# B&R Automation Studio project Panasonic_LinkaKapacitorov_A2021040 (part 5)

#### Main.st - Init, cyclic, exit code
```iecst
PROGRAM _INIT
	(* Insert code here *)

END_PROGRAM

PROGRAM _CYCLIC

	//Volanie podprogramov//
	OvlCentrovacky;

	//Volanie funkcie SequenceControl//
	SequenceControl(SC:= SC_StoperDopravNG);

	//Príznak obsluha potvrdila paletku NG na dopravníku NG//
	IF StoperDopravNG.Automat AND StoperDopravNG.STAV.PaletkaNaKonciDopravnika_NG AND Vizu.TL_NavratPaletkyNG THEN
		StoperDopravNG.STAV.ObsluhaPotvrdilaPaletkuNG:= TRUE;
		Vizu.TL_NavratPaletkyNG:= FALSE;
	END_IF
	IF NOT StoperDopravNG.IN.Dopravnik_PritomnostPaletky_OS4 THEN
		StoperDopravNG.STAV.ObsluhaPotvrdilaPaletkuNG:= FALSE;
	END_IF

	//Zmena farby tlačítka potvrdenie návratu paletky NG//
	IF StoperDopravNG.STAV.ObsluhaPotvrdilaPaletkuNG THEN
		Vizu.FarbaTlacitka_PotvrdPaletkuNG:= Blikac500ms;
	ELSE
		Vizu.FarbaTlacitka_PotvrdPaletkuNG:= TRUE;
	END_IF

	//Zobrazenie hlásenia potvrd paletku NG//
	IF StoperDopravNG.STAV.PaletkaNaKonciDopravnika_NG AND NOT StoperDopravNG.STAV.DopravnikNG_BUSY AND StoperDopravNG.STAV.PoINIT THEN
		Vizu.ZobrazHlasenie_PotvrdPaletkyNG:= 0;
	ELSE
		Vizu.ZobrazHlasenie_PotvrdPaletkyNG:= 1;
	END_IF

	//Príznak paletka NG na konci dopravníka//
	IF StoperDopravNG.Automat AND StoperDopravNG.IN.Dopravnik_PritomnostPaletky_OS4 THEN
		StoperDopravNG.STAV.PaletkaNaKonciDopravnika_NG:= TRUE;
	END_IF

	//Zamknutie tlačítka potvrdenie paletky NG//
	IF StoperDopravNG.STAV.PaletkaNaKonciDopravnika_NG AND StoperDopravNG.IN.Dopravnik_PritomnostPaletky_OS4 THEN
		Vizu.TL_PotvrdeniePaletky_NG_DISABLE:= FALSE;
	ELSE
		Vizu.TL_PotvrdeniePaletky_NG_DISABLE:= TRUE;
	END_IF

	//Zamknutie tlačítka zrušenie paletky NG//
	IF StoperDopravNG.STAV.PaletkaNaKonciDopravnika_NG AND NOT StoperDopravNG.IN.Dopravnik_PritomnostPaletky_OS4 THEN
		Vizu.TL_ZruseniePaletky_NG_DISABLE:= FALSE;
	ELSE
		Vizu.TL_ZruseniePaletky_NG_DISABLE:= TRUE;
	END_IF

	//Zrušenie paletky NG//
	IF StoperDopravNG.STAV.ObsluhaPotvrdilaZrusPaletkyNG THEN
		StoperDopravNG.STAV.PaletkaNaKonciDopravnika_NG:= FALSE;
		StoperDopravNG.STAV.ObsluhaPotvrdilaZrusPaletkyNG:= FALSE;
	END_IF

	//Reset sekcie //
	IF StoperDopravNG.Reset THEN
		SC_StoperDopravNG.Step:= 0;
		StoperDopravNG.Reset:= FALSE;
	ELSIF NOT Safety.STAV.ZonaCS_AKTIVNA THEN
		SC_StoperDopravNG.Step:= 0;
	END_IF

	CASE SC_StoperDopravNG.Step OF

		0:
			SC_StoperDopravNG.StepName:='0 - Nulovanie';
			StoperDopravNG.Automat:= FALSE;
			StoperDopravNG.KoniecCyklu:= FALSE;
			StoperDopravNG.Manual:= FALSE;
			StoperDopravNG.STAV.PoINIT:= FALSE;
			StoperDopravNG.OUT.Dopravnik_ChodVPRED_ELR3:= FALSE;
			StoperDopravNG.OUT.Dopravnik_ChodVZAD_ELR3:= FALSE;
			SC_OvlCentrovacky.Step:= 0;
			StoperDopravNG.STAV.ObsluhaPotvrdilaPaletkuNG:= FALSE;
			StoperDopravNG.RR_Dopravnik_VPRED:= FALSE;
			StoperDopravNG.RR_Dopravnik_VZAD:= FALSE;
			Vizu.ZobrazHlasenie_PotvrdPaletkyNG:= 1;
			StoperDopravNG.STAV.PrebiehaVyvazaniePaletky:= FALSE;
			StoperDopravNG.STAV.PaletkaNaKonciDopravnika_NG:= FALSE;
			StoperDopravNG.STAV.DopravnikNG_BUSY:= FALSE;
			StoperDopravNG_Statistika.IN.START_MeraniaCasu:= FALSE;

			IF Safety.STAV.ZonaCS_AKTIVNA AND Safety.STAV.ZonaBunky_AKTIVNA AND Linka.IN.TlakVzduchu_OK_S2 AND NOT NastalaPorucha AND Linka.STAV.Hardware_OK THEN
				SC_StoperDopravNG.ResetStep:= TRUE;
				SC_StoperDopravNG.Step:= 1;
			END_IF

		1:
			SC_StoperDopravNG.StepName:='1 - Cakam na spustenie vyroby';
			StoperDopravNG.KoniecCyklu:= FALSE;
			IF StoperDopravNG.Automat THEN
				SC_StoperDopravNG.Step:= 2;
			ELSIF StoperDopravNG.Manual THEN
				SC_StoperDopravNG.Step:= 700;
			END_IF

			//********************************************************Inicializácia****************************************************************************//

		2:
			SC_StoperDopravNG.StepName:='2 - Inicializacia - cakam na spustenie inicializacie';
			SC_StoperDopravNG.IdleTime.PT:= T#4s;
			SC_StoperDopravNG.AlarmTime.PT:= T#5s;

			IF DopravBunky.STAV.PoINIT AND Robot.STAV.PoINIT THEN
				SC_StoperDopravNG.ResetStep:= TRUE;
				SC_StoperDopravNG.Step:= 5;
			END_IF

		5:
			SC_StoperDopravNG.StepName:='5 - Inicializacia - hladanie paletky na dopravniku NG';
			SC_StoperDopravNG.IdleTime.PT:= T#5s;
			SC_StoperDopravNG.AlarmTime.PT:= T#5s;

			IF NOT SC_StoperDopravNG.Switch1 AND Safety.STAV.MutingRobota_AKTIVNY THEN
				StoperDopravNG.OUT.Dopravnik_ChodVPRED_ELR3:= TRUE;
				StoperDopravNG.STAV.DopravnikNG_BUSY:= TRUE;
				SC_StoperDopravNG.IdleTime.IN:= TRUE;
				SC_StoperDopravNG.Switch1:= TRUE;
			END_IF

			IF StoperDopravNG.IN.Dopravnik_PritomnostPaletky_OS4 THEN
				StoperDopravNG.OUT.Dopravnik_ChodVPRED_ELR3:= FALSE;
				StoperDopravNG.STAV.DopravnikNG_BUSY:= FALSE;
				Vizu.ZobrazHlasenie_PotvrdPaletkyNG:= 0;
				SC_StoperDopravNG.ResetStep:= TRUE;
				SC_StoperDopravNG.Step:= 10;
			ELSIF SC_StoperDopravNG.IdleTime.Q THEN
				StoperDopravNG.OUT.Dopravnik_ChodVPRED_ELR3:= FALSE;
				StoperDopravNG.STAV.DopravnikNG_BUSY:= FALSE;
				SC_StoperDopravNG.ResetStep:= TRUE;
				SC_StoperDopravNG.Step:= 10;
			END_IF

		10:
			SC_StoperDopravNG.StepName:='10 - Inicializacia - presun centrovacky do sterdnej polohy';
			SC_StoperDopravNG.IdleTime.PT:= T#4s;
			SC_StoperDopravNG.AlarmTime.PT:= T#5s;

			IF NOT SC_StoperDopravNG.Switch1 THEN
				Centrovacku_VYSTRED:= TRUE;
				SC_StoperDopravNG.Switch1:= TRUE;
			END_IF

			IF StoperDopravNG.IN.Centrovanie_StrednaPoloha_IS20 THEN
				SC_StoperDopravNG.ResetStep:= TRUE;
				SC_StoperDopravNG.Step:= 13;
			END_IF

		13:
			SC_StoperDopravNG.StepName:='13 - Inicializacia - hladanie paletky';
			SC_StoperDopravNG.IdleTime.PT:= T#3s;
			SC_StoperDopravNG.AlarmTime.PT:= T#7s;

			SC_StoperDopravNG.IdleTime.IN:= StoperDopravNG.IN.Stoper_PritomnostPaletky_IS15;
			SC_StoperDopravNG.AlarmTime.IN:= TRUE;

			IF SC_StoperDopravNG.IdleTime.Q THEN
				StoperDopravNG.STAV.PoINIT:= TRUE;
				SC_StoperDopravNG.ResetStep:= TRUE;
				SC_StoperDopravNG.Step:= 100;
			ELSIF SC_StoperDopravNG.AlarmTime.Q AND NOT StoperDopravNG.IN.Stoper_PritomnostPaletky_IS15 THEN
				StoperDopravNG.STAV.PoINIT:= TRUE;
				SC_StoperDopravNG.ResetStep:= TRUE;
				SC_StoperDopravNG.Step:= 100;
			END_IF

			//********************************************************Automatický režim****************************************************************************//

		100:
			SC_StoperDopravNG.StepName:='100 - Automaticky Rezim - cakam na príchod paletky na stoper';
			SC_StoperDopravNG.IdleTime.PT:= T#3s;
			SC_StoperDopravNG.AlarmTime.PT:= T#5s;

			SC_StoperDopravNG.IdleTime.IN:= StoperDopravNG.IN.Stoper_PritomnostPaletky_IS15;

			IF StoperDopravNG.KoniecCyklu THEN
				SC_StoperDopravNG.ResetStep:= TRUE;
				SC_StoperDopravNG.Step:= 0;
			ELSIF SC_StoperDopravNG.IdleTime.Q THEN
				StoperDopravNG_Statistika.IN.START_MeraniaCasu:= TRUE;
				StoperDopravNG_Statistika.IN.ZAPIS_MeraniaCasu:= TRUE;
				SC_StoperDopravNG.ResetStep:= TRUE;
				SC_StoperDopravNG.Step:= 110;
			ELSIF NOT StoperDopravNG.IN.Stoper_PritomnostPaletky_IS15 AND StoperDopravNG.IN.Dopravnik_PritomnostPaletky_OS4 AND NOT StoperEtiketovania.STAV.PrebiehaVyvazaniePaletky AND StoperDopravNG.STAV.ObsluhaPotvrdilaPaletkuNG AND NOT StoperEtiketovania.STAV.Etiketovanie_BUSY AND NOT StoperVystupDopravnika.IN.ZaplnenieBuffera_IS28 THEN
				StoperDopravNG.STAV.DopravnikNG_BUSY:= TRUE;
				SC_StoperDopravNG.ResetStep:= TRUE;
				SC_StoperDopravNG.Step:= 150;
			END_IF

		110:
			SC_StoperDopravNG.StepName:='110 - Automaticky Rezim - kontrola stavu paletky';
			SC_StoperDopravNG.IdleTime.PT:= T#200ms;
			SC_StoperDopravNG.AlarmTime.PT:= T#10s;

			IF StoperEtiketovania.STAV.VyvazamPaletkuNG THEN
				StoperDopravNG.STAV.DopravnikNG_BUSY:= TRUE;
				SC_StoperDopravNG.ResetStep:= TRUE;
				SC_StoperDopravNG.Step:= 120;
			ELSE
				SC_StoperDopravNG.ResetStep:= TRUE;
				SC_StoperDopravNG.Step:= 170;
			END_IF

			//Vyvezenie na dopravník NG//
		120:
			SC_StoperDopravNG.StepName:='120 - Automaticky Rezim - kontrola muting pozicie robota';
			SC_StoperDopravNG.IdleTime.PT:= T#200ms;
			SC_StoperDopravNG.AlarmTime.PT:= T#10s;

			IF Safety.STAV.MutingRobota_AKTIVNY AND Robot.STAV.PoINIT THEN
				SC_StoperDopravNG.ResetStep:= TRUE;
				SC_StoperDopravNG.Step:= 128;
			ELSIF NOT Safety.STAV.MutingRobota_AKTIVNY AND Robot.STAV.PoINIT THEN
				Robot.KOM_OUT.PresunDoMutingPozicie:= TRUE;
				SC_StoperDopravNG.ResetStep:= TRUE;
				SC_StoperDopravNG.Step:= 123;
			END_IF

		123:
			SC_StoperDopravNG.StepName:='123 - Automaticky Rezim - cakam na ukoncenie cinnosti robota';
			SC_StoperDopravNG.IdleTime.PT:= T#200ms;
			SC_StoperDopravNG.AlarmTime.PT:= T#10s;

			IF Robot.KOM_IN.Stav_RobotCinnostUkoncena THEN
				Robot.KOM_OUT.PresunDoMutingPozicie:= FALSE;
				SC_StoperDopravNG.ResetStep:= TRUE;
				SC_StoperDopravNG.Step:= 125;
			END_IF

		125:
			SC_StoperDopravNG.StepName:='125 - Automaticky Rezim - cakam na zrusenie signalu cinnost robota ukoncena';
			SC_StoperDopravNG.IdleTime.PT:= T#200ms;
			SC_StoperDopravNG.AlarmTime.PT:= T#5s;

			IF NOT Robot.KOM_IN.Stav_RobotCinnostUkoncena AND Safety.STAV.MutingRobota_AKTIVNY THEN
				SC_StoperDopravNG.ResetStep:= TRUE;
				SC_StoperDopravNG.Step:= 128;
			END_IF

		128:
			SC_StoperDopravNG.StepName:='128 - Automaticky Rezim - zdvih centrovacky pre vyvezenie paletky na dopravnik NG';
			SC_StoperDopravNG.IdleTime.PT:= T#200ms;
			SC_StoperDopravNG.AlarmTime.PT:= T#10s;

			IF NOT SC_StoperDopravNG.Switch1 THEN
				Centrovacku_VYSUN:= TRUE;
				SC_StoperDopravNG.Switch1:= TRUE;
			END_IF

			IF StoperDopravNG.IN.Centrovanie_HornaPoloha_IS19 THEN
				SC_StoperDopravNG.ResetStep:= TRUE;
				SC_StoperDopravNG.Step:= 130;
			END_IF

		130:
			SC_StoperDopravNG.StepName:='130 - Automaticky Rezim - spustenie dopravnika NG vpred';
			SC_StoperDopravNG.IdleTime.PT:= T#200ms;
			SC_StoperDopravNG.AlarmTime.PT:= T#10s;

			SC_StoperDopravNG.IdleTime.IN:= StoperDopravNG.IN.Dopravnik_PritomnostPaletky_OS4;

			IF NOT SC_StoperDopravNG.Switch1 AND Safety.STAV.MutingRobota_AKTIVNY THEN
				StoperDopravNG.OUT.Dopravnik_ChodVPRED_ELR3:= TRUE;
				SC_StoperDopravNG.AlarmTime.IN:= TRUE;
				SC_StoperDopravNG.Switch1:= TRUE;
			END_IF

			IF SC_StoperDopravNG.IdleTime.Q THEN
				(*StoperDopravNG.OUT.Dopravnik_ChodVPRED_ELR3:= FALSE;*)
				StoperDopravNG.STAV.PaletkaNaKonciDopravnika_NG:= TRUE;
				StoperDopravNG.STAV.DopravnikNG_BUSY:= FALSE;
				Vizu.ZobrazHlasenie_PotvrdPaletkyNG:= 0;
				SC_StoperDopravNG.ResetStep:= TRUE;
				SC_StoperDopravNG.Step:= 133;
			ELSIF SC_StoperDopravNG.AlarmTime.Q THEN
				Alarmy[63]:= TRUE;
				PoruchaBunky:= TRUE;
				SC_StoperDopravNG.ResetStep:= TRUE;
				SC_StoperDopravNG.Step:= 0;
			END_IF

		133:
			SC_StoperDopravNG.StepName:='133 - Automaticky Rezim - presun centrovacky do strednej polohy';
			SC_StoperDopravNG.IdleTime.PT:= T#4s;
			SC_StoperDopravNG.AlarmTime.PT:= T#5s;

			IF NOT SC_StoperDopravNG.Switch1 THEN
				Centrovacku_VYSTRED:= TRUE;
				SC_StoperDopravNG.Switch1:= TRUE;
			END_IF

			IF StoperDopravNG.IN.Centrovanie_StrednaPoloha_IS20 THEN
				SC_StoperDopravNG.ResetStep:= TRUE;
				SC_StoperDopravNG.Step:= 100;
			END_IF

			//Navezenie z dopravníka NG//
		150:
			SC_StoperDopravNG.StepName:='150 - Automaticky Rezim - kontrola muting pozicie robota';
			SC_StoperDopravNG.IdleTime.PT:= T#200ms;
			SC_StoperDopravNG.AlarmTime.PT:= T#10s;

			IF Safety.STAV.MutingRobota_AKTIVNY THEN
				SC_StoperDopravNG.ResetStep:= TRUE;
				SC_StoperDopravNG.Step:= 158;
			ELSIF NOT Safety.STAV.MutingRobota_AKTIVNY AND Robot.Automat THEN
				Robot.KOM_OUT.PresunDoMutingPozicie:= TRUE;
				SC_StoperDopravNG.ResetStep:= TRUE;
				SC_StoperDopravNG.Step:= 153;
			END_IF

		153:
			SC_StoperDopravNG.StepName:='153 - Automaticky Rezim - cakam na ukoncenie cinnosti robota';
			SC_StoperDopravNG.IdleTime.PT:= T#200ms;
			SC_StoperDopravNG.AlarmTime.PT:= T#10s;

			IF Robot.KOM_IN.Stav_RobotCinnostUkoncena THEN
				Robot.KOM_OUT.PresunDoMutingPozicie:= FALSE;
				SC_StoperDopravNG.ResetStep:= TRUE;
				SC_StoperDopravNG.Step:= 155;
			END_IF

		155:
			SC_StoperDopravNG.StepName:='155 - Automaticky Rezim - cakam na zrusenie signalu cinnost robota ukoncena';
			SC_StoperDopravNG.IdleTime.PT:= T#200ms;
			SC_StoperDopravNG.AlarmTime.PT:= T#5s;

			IF NOT Robot.KOM_IN.Stav_RobotCinnostUkoncena AND Safety.STAV.MutingRobota_AKTIVNY THEN
				SC_StoperDopravNG.ResetStep:= TRUE;
				SC_StoperDopravNG.Step:= 158;
			END_IF

		158:
			SC_StoperDopravNG.StepName:='150 - Automaticky Rezim - zdvih centrovacky pre navezenie paletky z dopravnika NG';
			SC_StoperDopravNG.IdleTime.PT:= T#200ms;
			SC_StoperDopravNG.AlarmTime.PT:= T#10s;

			IF NOT SC_StoperDopravNG.Switch1 THEN
				Centrovacku_VYSUN:= TRUE;
				SC_StoperDopravNG.Switch1:= TRUE;
			END_IF

			IF StoperDopravNG.IN.Centrovanie_HornaPoloha_IS19 THEN
				SC_StoperDopravNG.ResetStep:= TRUE;
				SC_StoperDopravNG.Step:= 160;
			END_IF

		160:
			SC_StoperDopravNG.StepName:='160 - Automaticky Rezim - spustenie dopravnika NG vzad';
			SC_StoperDopravNG.IdleTime.PT:= T#200ms;
			SC_StoperDopravNG.AlarmTime.PT:= T#10s;

			SC_StoperDopravNG.IdleTime.IN:= StoperDopravNG.IN.Stoper_PritomnostPaletky_IS15;

			IF NOT SC_StoperDopravNG.Switch1 AND Safety.STAV.MutingRobota_AKTIVNY THEN
				StoperDopravNG.OUT.Dopravnik_ChodVPRED_ELR3:= FALSE;
				StoperDopravNG.OUT.Dopravnik_ChodVZAD_ELR3:= TRUE;
				SC_StoperDopravNG.AlarmTime.IN:= TRUE;
				SC_StoperDopravNG.Switch1:= TRUE;
			END_IF

			IF SC_StoperDopravNG.IdleTime.Q THEN
				StoperDopravNG.STAV.PaletkaNaKonciDopravnika_NG:= FALSE;
				StoperDopravNG.OUT.Dopravnik_ChodVZAD_ELR3:= FALSE;
				StoperDopravNG.STAV.DopravnikNG_BUSY:= FALSE;
				SC_StoperDopravNG.ResetStep:= TRUE;
				SC_StoperDopravNG.Step:= 163;
			ELSIF SC_StoperDopravNG.AlarmTime.Q THEN
				Alarmy[64]:= TRUE;
				PoruchaBunky:= TRUE;
				SC_StoperDopravNG.ResetStep:= TRUE;
				SC_StoperDopravNG.Step:= 0;
			END_IF

		163:
			SC_StoperDopravNG.StepName:='163 - Automaticky Rezim - presun centrovacky do strednej polohy';
			SC_StoperDopravNG.IdleTime.PT:= T#4s;
			SC_StoperDopravNG.AlarmTime.PT:= T#5s;

			IF NOT SC_StoperDopravNG.Switch1 THEN
				Centrovacku_VYSTRED:= TRUE;
				SC_StoperDopravNG.Switch1:= TRUE;
			END_IF

			IF StoperDopravNG.IN.Centrovanie_StrednaPoloha_IS20 THEN
				SC_StoperDopravNG.ResetStep:= TRUE;
				SC_StoperDopravNG.Step:= 170;
			END_IF

			//Vyvezenie paletky na výstupný dopravník//
		170:
			SC_StoperDopravNG.StepName:='170 - Automaticky Rezim - cakam na vyvezenie na stoper vystupneho dopravnika';
			SC_StoperDopravNG.IdleTime.PT:= T#4s;
			SC_StoperDopravNG.AlarmTime.PT:= T#5s;

			IF StoperDopravNG.KoniecCyklu THEN
				SC_StoperDopravNG.ResetStep:= TRUE;
				SC_StoperDopravNG.Step:= 0;
			ELSIF NOT StoperVystupDopravnika.IN.ZaplnenieBuffera_IS28 AND VystupnyDopravnik.STAV.PoINIT THEN
				SC_StoperDopravNG.ResetStep:= TRUE;
				SC_StoperDopravNG.Step:= 173;
			END_IF

		173:
			SC_StoperDopravNG.StepName:='173 - Automaticky Rezim - vyvazam paletku na stoper vystupneho dopravnika';
			SC_StoperDopravNG.IdleTime.PT:= T#500ms;
			SC_StoperDopravNG.AlarmTime.PT:= T#10s;

			SC_StoperDopravNG.IdleTime.IN:= NOT StoperDopravNG.IN.Stoper_PritomnostPaletky_IS15;

			IF NOT SC_StoperDopravNG.Switch1 THEN
				Centrovacku_ZASUN:= TRUE;
				StoperDopravNG.STAV.PrebiehaVyvazaniePaletky:= TRUE;
				SC_StoperDopravNG.AlarmTime.IN:= TRUE;
				SC_StoperDopravNG.Switch1:= TRUE;
			END_IF

			IF NOT SC_StoperDopravNG.Switch2 AND SC_StoperDopravNG.IdleTime.Q AND SC_OvlCentrovacky.Step = 1 THEN
				Centrovacku_VYSTRED:= TRUE;
				SC_StoperDopravNG.AlarmTime.IN:= FALSE;
				SC_StoperDopravNG.Switch2:= TRUE;
			END_IF

			IF NOT Linka.Rezim_Priechodny AND StoperDopravNG.IN.Centrovanie_StrednaPoloha_IS20 AND NOT StoperDopravNG.IN.Stoper_PritomnostPaletky_IS15 THEN
				StoperDopravNG.STAV.PrebiehaVyvazaniePaletky:= FALSE;
				SC_StoperDopravNG.ResetStep:= TRUE;
				SC_StoperDopravNG.Step:= 100;
			ELSIF Linka.Rezim_Priechodny AND StoperDopravNG.IN.Centrovanie_StrednaPoloha_IS20 AND NOT StoperDopravNG.IN.Stoper_PritomnostPaletky_IS15 AND StoperVystupDopravnika.IN.ZaplnenieBuffera_IS28 THEN
				StoperDopravNG.STAV.PrebiehaVyvazaniePaletky:= FALSE;
				SC_StoperDopravNG.ResetStep:= TRUE;
				SC_StoperDopravNG.Step:= 100;
			ELSIF SC_StoperDopravNG.AlarmTime.Q THEN
				Alarmy[65]:= TRUE;
				PoruchaBunky:= TRUE;
				SC_StoperDopravNG.ResetStep:= TRUE;
				SC_StoperDopravNG.Step:= 0;
			END_IF

			//*******************************************************Manuálny režim*******************************************************************************//
		700:
			SC_StoperDopravNG.StepName:='700 - Manualny Rezim';
			SC_StoperDopravNG.IdleTime.PT:= T#8s;
			SC_StoperDopravNG.AlarmTime.PT:= T#5s;

			//Ovládanie dopravníka//
			IF StoperDopravNG.RR_Dopravnik_VPRED THEN
				StoperDopravNG.RR_Dopravnik_VZAD:= FALSE;
				StoperDopravNG.OUT.Dopravnik_ChodVZAD_ELR3:= FALSE;
				StoperDopravNG.OUT.Dopravnik_ChodVPRED_ELR3:= TRUE;
			ELSIF StoperDopravNG.RR_Dopravnik_VZAD THEN
				StoperDopravNG.RR_Dopravnik_VPRED:= FALSE;
				StoperDopravNG.OUT.Dopravnik_ChodVPRED_ELR3:= FALSE;
				StoperDopravNG.OUT.Dopravnik_ChodVZAD_ELR3:= TRUE;
			ELSE
				StoperDopravNG.OUT.Dopravnik_ChodVPRED_ELR3:= FALSE;
				StoperDopravNG.OUT.Dopravnik_ChodVZAD_ELR3:= FALSE;
			END_IF

	END_CASE

END_PROGRAM

PROGRAM _EXIT
	(* Insert code here *)

END_PROGRAM
```

#### Variables.var - Local variables
```iecst
VAR
	SC_OvlCentrovacky : SequenceControlTyp;
	Centrovacku_VYSUN : BOOL;
	Centrovacku_ZASUN : BOOL;
	Centrovacku_VYSTRED : BOOL := FALSE;
END_VAR
```

#### OvlCentrovacky.st
```iecst
ACTION OvlCentrovacky:

	//Volanie funkcie SequenceControl//
	SequenceControl(SC:= SC_OvlCentrovacky);

	CASE SC_OvlCentrovacky.Step OF

		0:
			SC_OvlCentrovacky.StepName:= '0 - Nulovanie';
			Centrovacku_VYSUN:= FALSE;
			Centrovacku_ZASUN:= FALSE;
			Centrovacku_VYSTRED:= FALSE;
			//			StoperDopravNG.OUT.Centrovanie_VYSUN_YV009:= FALSE;
			//			StoperDopravNG.OUT.Centrovanie_ZASUN_YV010:= FALSE;

			IF SC_StoperDopravNG.Step <> 0 THEN
				SC_OvlCentrovacky.ResetStep:= TRUE;
				SC_OvlCentrovacky.Step:= 1;
			END_IF

		1:
			SC_OvlCentrovacky.StepName:= '1 - Rozhodnutie o cinnosti';
			IF Centrovacku_VYSUN THEN
				SC_OvlCentrovacky.Step:= 10;
			ELSIF Centrovacku_ZASUN THEN
				SC_OvlCentrovacky.Step:= 20;
			ELSIF Centrovacku_VYSTRED THEN
				SC_OvlCentrovacky.Step:= 30;
			END_IF

		10:
			SC_OvlCentrovacky.StepName:= '10 - Vysunutie centrovacky hore';
			SC_OvlCentrovacky.IdleTime.PT:= T#3s;
			SC_OvlCentrovacky.AlarmTime.PT:= T#6s;

			IF StoperDopravNG.Automat THEN
				SC_OvlCentrovacky.AlarmTime.IN:= TRUE;
			ELSE
				SC_OvlCentrovacky.IdleTime.IN:= TRUE;
			END_IF

			IF NOT SC_OvlCentrovacky.Switch1 THEN
				StoperDopravNG.OUT.Centrovanie_ZASUN_YV010:= FALSE;
				StoperDopravNG.OUT.Centrovanie_VYSUN_YV009:= TRUE;
				SC_OvlCentrovacky.Switch1:= TRUE;
			END_IF

			IF StoperDopravNG.IN.Centrovanie_HornaPoloha_IS19 OR SC_OvlCentrovacky.IdleTime.Q THEN
				SC_OvlCentrovacky.ResetStep:= TRUE;
				SC_OvlCentrovacky.Step:= 0;
			ELSIF SC_OvlCentrovacky.AlarmTime.Q THEN
				Alarmy[57]:= TRUE;
				PoruchaBunky:= TRUE;
				SC_OvlCentrovacky.ResetStep:= TRUE;
				SC_OvlCentrovacky.Step:= 0;
			END_IF

		20:
			SC_OvlCentrovacky.StepName:= '20 - Zasunutie centrovacky dole';
			SC_OvlCentrovacky.IdleTime.PT:= T#3s;
			SC_OvlCentrovacky.AlarmTime.PT:= T#6s;

			IF StoperDopravNG.Automat THEN
				SC_OvlCentrovacky.AlarmTime.IN:= TRUE;
			ELSE
				SC_OvlCentrovacky.IdleTime.IN:= TRUE;
			END_IF

			IF NOT SC_OvlCentrovacky.Switch1 THEN
				StoperDopravNG.OUT.Centrovanie_VYSUN_YV009:= FALSE;
				StoperDopravNG.OUT.Centrovanie_ZASUN_YV010:= TRUE;
				SC_OvlCentrovacky.Switch1:= TRUE;
			END_IF

			IF StoperDopravNG.IN.Centrovanie_SpodnaPoloha_IS21 OR SC_OvlCentrovacky.IdleTime.Q THEN
				SC_OvlCentrovacky.ResetStep:= TRUE;
				SC_OvlCentrovacky.Step:= 0;
			ELSIF SC_OvlCentrovacky.AlarmTime.Q THEN
				Alarmy[58]:= TRUE;
				PoruchaBunky:= TRUE;
				SC_OvlCentrovacky.ResetStep:= TRUE;
				SC_OvlCentrovacky.Step:= 0;
			END_IF

		30:
			SC_OvlCentrovacky.StepName:= '30 - Presun centrovacky do strednej polohy';
			SC_OvlCentrovacky.IdleTime.PT:= T#3s;
			SC_OvlCentrovacky.AlarmTime.PT:= T#6s;

			IF StoperDopravNG.Automat THEN
				SC_OvlCentrovacky.AlarmTime.IN:= TRUE;
			ELSE
				SC_OvlCentrovacky.IdleTime.IN:= TRUE;
			END_IF

			IF NOT SC_OvlCentrovacky.Switch1 THEN
				StoperDopravNG.OUT.Centrovanie_VYSUN_YV009:= FALSE;
				StoperDopravNG.OUT.Centrovanie_ZASUN_YV010:= FALSE;
				SC_OvlCentrovacky.Switch1:= TRUE;
			END_IF

			IF StoperDopravNG.IN.Centrovanie_StrednaPoloha_IS20 OR SC_OvlCentrovacky.IdleTime.Q THEN
				SC_OvlCentrovacky.ResetStep:= TRUE;
				SC_OvlCentrovacky.Step:= 0;
			ELSIF SC_OvlCentrovacky.AlarmTime.Q THEN
				Alarmy[59]:= TRUE;
				PoruchaBunky:= TRUE;
				SC_OvlCentrovacky.ResetStep:= TRUE;
				SC_OvlCentrovacky.Step:= 0;
			END_IF

	END_CASE

END_ACTION
```

### Program Logical/Program/DopravnikBunky (IEC)

#### Main.st - Init, cyclic, exit code
```iecst
PROGRAM _INIT
	(* Insert code here *)

END_PROGRAM

PROGRAM _CYCLIC

	//Volanie funkcie SequenceControl//
	SequenceControl(SC:= SC_DopravBunky);

	//Reset sekcie //
	IF DopravBunky.Reset THEN
		SC_DopravBunky.Step:= 0;
		DopravBunky.Reset:= FALSE;
	ELSIF NOT Safety.STAV.ZonaCS_AKTIVNA THEN
		SC_DopravBunky.Step:= 0;
	END_IF

	CASE SC_DopravBunky.Step OF

		0:
			SC_DopravBunky.StepName:='0 - Nulovanie';
			DopravBunky.Automat:= FALSE;
			DopravBunky.KoniecCyklu:= FALSE;
			DopravBunky.Manual:= FALSE;
			DopravBunky.STAV.PoINIT:= FALSE;
			DopravBunky.OUT.Dopravnik_ChodVPRED_ELR4:= FALSE;

			IF Safety.STAV.ZonaCS_AKTIVNA AND Safety.STAV.ZonaBunky_AKTIVNA  AND Linka.IN.TlakVzduchu_OK_S2 AND NOT NastalaPorucha AND Linka.STAV.Hardware_OK THEN
				SC_DopravBunky.ResetStep:= TRUE;
				SC_DopravBunky.Step:= 1;
			END_IF

		1:
			SC_DopravBunky.StepName:='1 - Cakam na spustenie vyroby';
			DopravBunky.KoniecCyklu:= FALSE;
			IF DopravBunky.Automat THEN
				SC_DopravBunky.Step:= 2;
			ELSIF DopravBunky.Manual THEN
				SC_DopravBunky.Step:= 700;
			END_IF

			//********************************************************Inicializácia****************************************************************************//

		2:
			SC_DopravBunky.StepName:='2 - Inicializacia - cakam na spustenie inicializacie';
			SC_DopravBunky.IdleTime.PT:= T#500ms;
			SC_DopravBunky.AlarmTime.PT:= T#5s;

			IF Robot.STAV.PoINIT THEN
				SC_DopravBunky.IdleTime.IN:= TRUE;
			END_IF

			IF SC_DopravBunky.IdleTime.Q THEN
				SC_DopravBunky.ResetStep:= TRUE;
				SC_DopravBunky.Step:= 5;
			END_IF

		5:
			SC_DopravBunky.StepName:='5 - Inicializacia - spustenie dopravnika a ukoncenie inicializacie';
			SC_DopravBunky.IdleTime.PT:= T#2s;
			SC_DopravBunky.AlarmTime.PT:= T#5s;

			IF NOT SC_DopravBunky.Switch1 THEN
				DopravBunky.OUT.Dopravnik_ChodVPRED_ELR4:= TRUE;
				SC_DopravBunky.IdleTime.IN:= TRUE;
				SC_DopravBunky.Switch1:= TRUE;
			END_IF

			IF SC_DopravBunky.IdleTime.Q THEN
				DopravBunky.STAV.PoINIT:= TRUE;
				SC_DopravBunky.ResetStep:= TRUE;
				SC_DopravBunky.Step:= 100;
			END_IF

			//********************************************************Automatický režim****************************************************************************//

		100:
			SC_DopravCistenia.StepName:='100 - Automaticky Rezim - cakam na vypnutie dopravnika';
			SC_DopravCistenia.IdleTime.PT:= T#5s;
			SC_DopravCistenia.AlarmTime.PT:= T#5s;

			SC_DopravCistenia.IdleTime.IN:= NOT StoperEtiketovania.Automat AND NOT StoperDopravNG.Automat AND NOT StoperPoCisteni.Automat;

			DopravBunky.OUT.Dopravnik_ChodVPRED_ELR4:= NOT Linka.STAV.Dopravniky_PAUZA;

			IF DopravBunky.KoniecCyklu AND SC_DopravCistenia.IdleTime.Q THEN
				SC_DopravBunky.ResetStep:= TRUE;
				SC_DopravBunky.Step:= 0;
			END_IF

			//*******************************************************Manuálny režim*******************************************************************************//
		700:
			SC_DopravBunky.StepName:='700 - Manualny Rezim';
			SC_DopravBunky.IdleTime.PT:= T#8s;
			SC_DopravBunky.AlarmTime.PT:= T#5s;

	END_CASE

END_PROGRAM

PROGRAM _EXIT
	(* Insert code here *)

END_PROGRAM
```

### Program Logical/Program/StoperVystupDopravnika (IEC)

#### Main.st - Init, cyclic, exit code
```iecst
PROGRAM _INIT
	(* Insert code here *)

END_PROGRAM

PROGRAM _CYCLIC

	//Volanie funkcie SequenceControl//
	SequenceControl(SC:= SC_StoperVystupDopravnika);

	//Reset sekcie //
	IF StoperVystupDopravnika.Reset THEN
		SC_StoperVystupDopravnika.Step:= 0;
		StoperVystupDopravnika.Reset:= FALSE;
	ELSIF NOT Safety.STAV.ZonaCS_AKTIVNA THEN
		SC_StoperVystupDopravnika.Step:= 0;
	END_IF

	CASE SC_StoperVystupDopravnika.Step OF

		0:
			SC_StoperVystupDopravnika.StepName:='0 - Nulovanie';
			StoperVystupDopravnika.Automat:= FALSE;
			StoperVystupDopravnika.KoniecCyklu:= FALSE;
			StoperVystupDopravnika.Manual:= FALSE;
			StoperVystupDopravnika.STAV.PoINIT:= FALSE;
			StoperVystupDopravnika.OUT.StoperZASUN_YV011:= FALSE;
			StoperVystupDopravnika.STAV.PrebiehaVyvazaniePaletky:= FALSE;

			IF Safety.STAV.ZonaCS_AKTIVNA AND Linka.IN.TlakVzduchu_OK_S2 AND NOT NastalaPorucha AND Linka.STAV.Hardware_OK THEN
				SC_StoperVystupDopravnika.ResetStep:= TRUE;
				SC_StoperVystupDopravnika.Step:= 1;
			END_IF

		1:
			SC_StoperVystupDopravnika.StepName:='1 - Cakam na spustenie vyroby';
			StoperVystupDopravnika.KoniecCyklu:= FALSE;
			IF StoperVystupDopravnika.Automat THEN
				SC_StoperVystupDopravnika.Step:= 2;
			ELSIF StoperVystupDopravnika.Manual THEN
				SC_StoperVystupDopravnika.Step:= 700;
			END_IF

			//********************************************************Inicializácia****************************************************************************//

		2:
			SC_StoperVystupDopravnika.StepName:='2 - Inicializacia - cakam na spustenie inicializacie';
			SC_StoperVystupDopravnika.IdleTime.PT:= T#4s;
			SC_StoperVystupDopravnika.AlarmTime.PT:= T#5s;

			IF VystupnyDopravnik.STAV.PoINIT THEN
				SC_StoperVystupDopravnika.ResetStep:= TRUE;
				SC_StoperVystupDopravnika.Step:= 3;
			END_IF

		3:
			SC_StoperVystupDopravnika.StepName:='3 - Inicializacia - hladanie paletky';
			SC_StoperVystupDopravnika.IdleTime.PT:= T#5s;
			SC_StoperVystupDopravnika.AlarmTime.PT:= T#5s;
			SC_StoperVystupDopravnika.IdleTime.IN:= TRUE;

			IF StoperVystupDopravnika.IN.PritomnostPaletky_IS27 THEN
				StoperVystupDopravnika.STAV.PoINIT:= TRUE;
				SC_StoperVystupDopravnika.ResetStep:= TRUE;
				SC_StoperVystupDopravnika.Step:= 101;
			ELSIF SC_StoperVystupDopravnika.IdleTime.Q THEN
				StoperVystupDopravnika.STAV.PoINIT:= TRUE;
				SC_StoperVystupDopravnika.ResetStep:= TRUE;
				SC_StoperVystupDopravnika.Step:= 100;
			END_IF

			//********************************************************Automatický režim****************************************************************************//
		100:
			SC_StoperVystupDopravnika.StepName:='100 - Automaticky Rezim - cakam na príchod paletky na stoper';
			SC_StoperVystupDopravnika.IdleTime.PT:= T#200ms;
			SC_StoperVystupDopravnika.AlarmTime.PT:= T#5s;

			SC_StoperVystupDopravnika.IdleTime.IN:= StoperVystupDopravnika.IN.PritomnostPaletky_IS27;

			IF StoperVystupDopravnika.KoniecCyklu THEN
				SC_StoperVystupDopravnika.ResetStep:= TRUE;
				SC_StoperVystupDopravnika.Step:= 0;
			ELSIF SC_StoperVystupDopravnika.IdleTime.Q THEN
				SC_StoperVystupDopravnika.ResetStep:= TRUE;
				SC_StoperVystupDopravnika.Step:= 101;
			END_IF

		101:
			SC_StoperVystupDopravnika.StepName:='101 - Automaticky Rezim - cakam na vyvezenie paletky na dopravnik vystupneho vytahu';
			SC_StoperVystupDopravnika.IdleTime.PT:= T#200ms;
			SC_StoperVystupDopravnika.AlarmTime.PT:= T#5s;

			IF StoperVystupDopravnika.KoniecCyklu THEN
				SC_StoperVystupDopravnika.ResetStep:= TRUE;
				SC_StoperVystupDopravnika.Step:= 0;
			ELSIF SC_VystupVytah.Step = 100 AND NOT VystupVytah.IN.PritomnostPaletky_IS26 THEN
				SC_StoperVystupDopravnika.ResetStep:= TRUE;
				SC_StoperVystupDopravnika.Step:= 105;
			END_IF

		105:
			SC_StoperVystupDopravnika.StepName:='105 - Automaticky Rezim - vyvazam paletku na dopravnik vystupneho vytahu';
			SC_StoperVystupDopravnika.IdleTime.PT:= T#4s;
			SC_StoperVystupDopravnika.AlarmTime.PT:= T#10s;

			IF NOT SC_StoperVystupDopravnika.Switch1 THEN
				StoperVystupDopravnika.OUT.StoperZASUN_YV011:= TRUE;
				StoperVystupDopravnika.STAV.PrebiehaVyvazaniePaletky:= TRUE;
				SC_StoperVystupDopravnika.AlarmTime.IN:= TRUE;
				SC_StoperVystupDopravnika.Switch1:= TRUE;
			END_IF

			IF NOT StoperVystupDopravnika.IN.PritomnostPaletky_IS27 THEN
				StoperVystupDopravnika.OUT.StoperZASUN_YV011:= FALSE;
				SC_StoperVystupDopravnika.AlarmTime.IN:= FALSE;
			END_IF

			IF VystupVytah.IN.PritomnostPaletky_IS26 AND NOT StoperVystupDopravnika.OUT.StoperZASUN_YV011  THEN
				StoperVystupDopravnika.STAV.PrebiehaVyvazaniePaletky:= FALSE;
				SC_StoperVystupDopravnika.ResetStep:= TRUE;
				SC_StoperVystupDopravnika.Step:= 100;
			ELSIF SC_StoperVystupDopravnika.AlarmTime.Q THEN
				Alarmy[40]:= TRUE;
				PoruchaVystupnehoVytahu:= TRUE;
				SC_StoperVystupDopravnika.ResetStep:= TRUE;
				SC_StoperVystupDopravnika.Step:= 0;
			END_IF

			//*******************************************************Manuálny režim*******************************************************************************//
		700:
			SC_StoperVystupDopravnika.StepName:='700 - Manualny Rezim';
			SC_StoperVystupDopravnika.IdleTime.PT:= T#8s;
			SC_StoperVystupDopravnika.AlarmTime.PT:= T#5s;

	END_CASE

END_PROGRAM

PROGRAM _EXIT
	(* Insert code here *)

END_PROGRAM
```

### Program Logical/Program/VystupnyDopravnik (IEC)

#### Main.st - Init, cyclic, exit code
```iecst
PROGRAM _INIT
	(* Insert code here *)

END_PROGRAM

PROGRAM _CYCLIC

	//Volanie funkcie SequenceControl//
	SequenceControl(SC:= SC_VystupnyDopravnik);

	//Reset sekcie //
	IF VystupnyDopravnik.Reset THEN
		SC_VystupnyDopravnik.Step:= 0;
		VystupnyDopravnik.Reset:= FALSE;
	ELSIF NOT Safety.STAV.ZonaCS_AKTIVNA THEN
		SC_VystupnyDopravnik.Step:= 0;
	END_IF

	CASE SC_VystupnyDopravnik.Step OF

		0:
			SC_VystupnyDopravnik.StepName:='0 - Nulovanie';
			VystupnyDopravnik.Automat:= FALSE;
			VystupnyDopravnik.KoniecCyklu:= FALSE;
			VystupnyDopravnik.Manual:= FALSE;
			VystupnyDopravnik.STAV.PoINIT:= FALSE;
			VystupnyDopravnik.OUT.Dopravnik_ChodVPRED_ELR5:= FALSE;

			IF Safety.STAV.ZonaCS_AKTIVNA AND Linka.IN.TlakVzduchu_OK_S2 AND NOT NastalaPorucha AND Linka.STAV.Hardware_OK THEN
				SC_VystupnyDopravnik.ResetStep:= TRUE;
				SC_VystupnyDopravnik.Step:= 1;
			END_IF

		1:
			SC_VystupnyDopravnik.StepName:='1 - Cakam na spustenie vyroby';
			VystupnyDopravnik.KoniecCyklu:= FALSE;
			IF VystupnyDopravnik.Automat THEN
				SC_VystupnyDopravnik.Step:= 2;
			ELSIF VystupnyDopravnik.Manual THEN
				SC_VystupnyDopravnik.Step:= 700;
			END_IF

			//********************************************************Inicializácia****************************************************************************//

		2:
			SC_VystupnyDopravnik.StepName:='2 - Inicializacia - cakam na spustenie inicializacie';
			SC_VystupnyDopravnik.IdleTime.PT:= T#500ms;
			SC_VystupnyDopravnik.AlarmTime.PT:= T#5s;

			SC_VystupnyDopravnik.IdleTime.IN:= TRUE;

			IF SC_VystupnyDopravnik.IdleTime.Q THEN
				SC_VystupnyDopravnik.ResetStep:= TRUE;
				SC_VystupnyDopravnik.Step:= 5;
			END_IF

		5:
			SC_VystupnyDopravnik.StepName:='5 - Inicializacia - spustenie dopravnika a ukoncenie inicializacie';
			SC_VystupnyDopravnik.IdleTime.PT:= T#2s;
			SC_VystupnyDopravnik.AlarmTime.PT:= T#5s;

			IF NOT SC_VystupnyDopravnik.Switch1 THEN
				VystupnyDopravnik.OUT.Dopravnik_ChodVPRED_ELR5:= TRUE;
				SC_VystupnyDopravnik.IdleTime.IN:= TRUE;
				SC_VystupnyDopravnik.Switch1:= TRUE;
			END_IF

			IF SC_VystupnyDopravnik.IdleTime.Q THEN
				VystupnyDopravnik.STAV.PoINIT:= TRUE;
				SC_VystupnyDopravnik.ResetStep:= TRUE;
				SC_VystupnyDopravnik.Step:= 100;
			END_IF

			//********************************************************Automatický režim****************************************************************************//

		100:
			SC_VystupnyDopravnik.StepName:='100 - Automaticky Rezim - cakam na vypnutie dopravnika';
			SC_VystupnyDopravnik.IdleTime.PT:= T#2s;
			SC_VystupnyDopravnik.AlarmTime.PT:= T#5s;

			SC_VystupnyDopravnik.IdleTime.IN:= NOT StoperVystupDopravnika.Automat AND NOT VystupVytah.Automat;

			VystupnyDopravnik.OUT.Dopravnik_ChodVPRED_ELR5:= NOT Linka.STAV.Dopravniky_PAUZA;

			IF VystupnyDopravnik.KoniecCyklu AND SC_VystupnyDopravnik.IdleTime.Q THEN
				SC_VystupnyDopravnik.ResetStep:= TRUE;
				SC_VystupnyDopravnik.Step:= 0;
			END_IF

			//*******************************************************Manuálny režim*******************************************************************************//
		700:
			SC_VystupnyDopravnik.StepName:='700 - Manualny Rezim';
			SC_VystupnyDopravnik.IdleTime.PT:= T#8s;
			SC_VystupnyDopravnik.AlarmTime.PT:= T#5s;

	END_CASE

END_PROGRAM

PROGRAM _EXIT
	(* Insert code here *)

END_PROGRAM
```

### Program Logical/Program/VystupnyVytah (IEC)

#### Main.st - Init, cyclic, exit code
```iecst
PROGRAM _INIT

	VystupVytah.PAR.Zdvih_ZadanaJoggRychlost:= 10;

END_PROGRAM

PROGRAM _CYCLIC

	//Volanie podprogramov//
	OvlMenica;
	OvlCitackyRFID;

	//Volanie funkcie SequenceControl//
	SequenceControl(SC:= SC_VystupVytah);

	//Reset sekcie //
	IF VystupVytah.Reset THEN
		SC_VystupVytah.Step:= 0;
		VystupVytah.Reset:= FALSE;
	ELSIF NOT Safety.STAV.ZonaCS_AKTIVNA THEN
		SC_VystupVytah.Step:= 0;
	END_IF

	CASE SC_VystupVytah.Step OF

		0:
			SC_VystupVytah.StepName:='0 - Nulovanie';
			VystupVytah.Automat:= FALSE;
			VystupVytah.KoniecCyklu:= FALSE;
			VystupVytah.Manual:= FALSE;
			VystupVytah.STAV.PoINIT:= FALSE;
			SC_OvlMenica.Step:= 0;
			VystupVytah.OUT.Dopravnik_ChodVPRED_ELR6:= FALSE;
			VystupVytah.OUT.Dopravnik_ChodVZAD_ELR6:= FALSE;
			VystupVytah.RR_Dopravnik_VPRED:= FALSE;
			VystupVytah.RR_Dopravnik_VZAD:= FALSE;
			VystupVytah.STAV.PrebiehaVyvazaniePaletky:= FALSE;
			IF PoruchaVystupnehoVytahu THEN
				VystupVytah.OUT.Banner_CervenaLED_IOS2:= Blikac200ms;
			ELSE
				VystupVytah.OUT.Banner_CervenaLED_IOS2:= FALSE;
			END_IF
			VystupVytah.OUT.Banner_ZelenaLED_IOS2:= FALSE;
			VystupVytah.STAV.VytahNapolohovany:= FALSE;
			VystupnyVytah_Statistika.IN.START_MeraniaCasu:= FALSE;

			IF Safety.STAV.ZonaCS_AKTIVNA AND Safety.STAV.ZonaVystupnyVytah_AKTIVNA AND Linka.IN.TlakVzduchu_OK_S2 AND NOT NastalaPorucha AND Linka.STAV.Hardware_OK THEN
				VystupVytah.OUT.Banner_CervenaLED_IOS2:= FALSE;
				SC_VystupVytah.ResetStep:= TRUE;
				SC_VystupVytah.Step:= 1;
			END_IF

		1:
			SC_VystupVytah.StepName:='1 - Cakam na spustenie vyroby';
			VystupVytah.KoniecCyklu:= FALSE;
			IF VystupVytah.Automat THEN
				SC_VystupVytah.Step:= 2;
			ELSIF VystupVytah.Manual THEN
				SC_VystupVytah.Step:= 700;
			END_IF

			//********************************************************Inicializácia****************************************************************************//

		2:
			SC_VystupVytah.StepName:='2 - Inicializacia - cakam na spustenie inicializacie';
			SC_VystupVytah.IdleTime.PT:= T#500ms;
			SC_VystupVytah.AlarmTime.PT:= T#5s;

			SC_VystupVytah.IdleTime.IN:= TRUE;

			IF SC_VystupVytah.IdleTime.Q THEN
				SC_VystupVytah.ResetStep:= TRUE;
				SC_VystupVytah.Step:= 5;
			END_IF

		5:
			SC_VystupVytah.StepName:='5 - Inicializacia - spustam dopravnik vytahu pre navezenie paletky';
			SC_VystupVytah.IdleTime.PT:= T#500ms;
			SC_VystupVytah.AlarmTime.PT:= T#7s;

			SC_VystupVytah.IdleTime.IN:= VystupVytah.IN.PritomnostPaletky_IS26;

			IF NOT SC_VystupVytah.Switch1 THEN
				VystupVytah.OUT.Dopravnik_ChodVPRED_ELR6:= TRUE;
				SC_VystupVytah.AlarmTime.IN:= TRUE;
				SC_VystupVytah.Switch1:= TRUE;
			END_IF

			IF SC_VystupVytah.IdleTime.Q AND NOT VystupVytah.IN.PrechodDopravnikaVytahu_OS6 THEN
				VystupVytah.OUT.Dopravnik_ChodVPRED_ELR6:= FALSE;
				SC_VystupVytah.ResetStep:= TRUE;
				SC_VystupVytah.Step:= 15;
			ELSIF SC_VystupVytah.AlarmTime.Q AND NOT VystupVytah.IN.PritomnostPaletky_IS26 AND NOT VystupVytah.IN.PrechodDopravnikaVytahu_OS6 THEN
				VystupVytah.OUT.Dopravnik_ChodVPRED_ELR6:= FALSE;
				SC_VystupVytah.ResetStep:= TRUE;
				SC_VystupVytah.Step:= 15;
			ELSIF SC_VystupVytah.AlarmTime.Q AND VystupVytah.IN.PrechodDopravnikaVytahu_OS6 THEN
				Alarmy[49]:= TRUE;
				PoruchaVystupnehoVytahu:= TRUE;
				SC_VystupVytah.ResetStep:= TRUE;
				SC_VystupVytah.Step:= 0;
			END_IF

		15:
			SC_VystupVytah.StepName:='15 - Inicializacia - kontrola homingu zdvihu vytahu';
			SC_VystupVytah.IdleTime.PT:= T#2s;
			SC_VystupVytah.AlarmTime.PT:= T#5s;

			IF VystupVytah.STAV.Zdvih_HomingOK THEN
				SC_VystupVytah.ResetStep:= TRUE;
				SC_VystupVytah.Step:= 35;
			ELSE
				SC_VystupVytah.ResetStep:= TRUE;
				SC_VystupVytah.Step:= 18;
			END_IF

		18:
			SC_VystupVytah.StepName:='18 - Inicializacia - cakam na spustenie homingu zdvihu vytahu';
			SC_VystupVytah.IdleTime.PT:= T#1s;
			SC_VystupVytah.AlarmTime.PT:= T#5s;

			SC_VystupVytah.IdleTime.IN:= Safety.STAV.BarieraVystupVytahu_AKTIVNA AND NOT VystupVytah.IN.PrechodDopravnikaVytahu_OS6;

			IF SC_VystupVytah.IdleTime.Q THEN
				SC_VystupVytah.ResetStep:= TRUE;
				SC_VystupVytah.Step:= 20;
			END_IF

		20:
			SC_VystupVytah.StepName:='20 - Inicializacia - spustam homing zdvihu vytahu';
			SC_VystupVytah.IdleTime.PT:= T#2s;
			SC_VystupVytah.AlarmTime.PT:= T#5s;

			VystupVytah.OUT.Banner_CervenaLED_IOS2:= TRUE;

			IF NOT SC_VystupVytah.Switch1 THEN
				Zdvih_HOME:= TRUE;
				SC_VystupVytah.Switch1:= TRUE;
			END_IF

			IF VystupVytah.STAV.Zdvih_HomingOK THEN
				SC_VystupVytah.ResetStep:= TRUE;
				SC_VystupVytah.Step:= 35;
			ELSIF NOT Safety.STAV.BarieraVystupVytahu_AKTIVNA THEN
				Alarmy[50]:= TRUE;
				PoruchaVystupnehoVytahu:= TRUE;
				SC_VystupVytah.ResetStep:= TRUE;
				SC_VystupVytah.Step:= 0;
			ELSIF VystupVytah.IN.PrechodDopravnikaVytahu_OS6 THEN
				Alarmy[51]:= TRUE;
				PoruchaVystupnehoVytahu:= TRUE;
				SC_VystupVytah.ResetStep:= TRUE;
				SC_VystupVytah.Step:= 0;
			END_IF

		35:
			SC_VystupVytah.StepName:='35 - Inicializacia - cakam na spustenie presunu vytahu do hornej pozicie navazania';
			SC_VystupVytah.IdleTime.PT:= T#1s;
			SC_VystupVytah.AlarmTime.PT:= T#5s;

			SC_VystupVytah.IdleTime.IN:= Safety.STAV.BarieraVystupVytahu_AKTIVNA AND NOT VystupVytah.IN.PrechodDopravnikaVytahu_OS6;

			IF SC_VystupVytah.IdleTime.Q THEN
				SC_VystupVytah.ResetStep:= TRUE;
				SC_VystupVytah.Step:= 38;
			END_IF

		38:
			SC_VystupVytah.StepName:='38 - Inicializacia - presuvam vytah do hornej pozicie navazania';
			SC_VystupVytah.IdleTime.PT:= T#2s;
			SC_VystupVytah.AlarmTime.PT:= T#5s;

			VystupVytah.OUT.Banner_CervenaLED_IOS2:= TRUE;
			VystupVytah.PAR.Zdvih_ZadanaRychlost:= 50;
			VystupVytah.PAR.Zdvih_ZadanaPozicia:= RemPremenne.VystupVytah_PozNavazania;

			IF NOT SC_VystupVytah.Switch1 AND SC_OvlMenica.Step = 1 THEN
				Zdvih_POLOHUJ:= TRUE;
				SC_VystupVytah.Switch1:= TRUE;
			END_IF

			IF VystupVytah.STAV.VytahNapolohovany THEN
				VystupVytah.STAV.VytahNapolohovany:= FALSE;
				VystupVytah.OUT.Banner_CervenaLED_IOS2:= FALSE;
				SC_VystupVytah.ResetStep:= TRUE;
				SC_VystupVytah.Step:= 40;
			ELSIF NOT Safety.STAV.BarieraVystupVytahu_AKTIVNA THEN
				Alarmy[50]:= TRUE;
				PoruchaVystupnehoVytahu:= TRUE;
				SC_VystupVytah.ResetStep:= TRUE;
				SC_VystupVytah.Step:= 0;
			ELSIF VystupVytah.IN.PrechodDopravnikaVytahu_OS6 THEN
				Alarmy[51]:= TRUE;
				PoruchaVystupnehoVytahu:= TRUE;
				SC_VystupVytah.ResetStep:= TRUE;
				SC_VystupVytah.Step:= 0;
			END_IF

		40:
			SC_VystupVytah.StepName:='40 - Inicializacia - kontrola pritomnosti paletky na dopravniku vytahu';
			SC_VystupVytah.IdleTime.PT:= T#2s;
			SC_VystupVytah.AlarmTime.PT:= T#5s;

			IF VystupVytah.IN.PritomnostPaletky_IS26 THEN
				VystupVytah.STAV.PoINIT := TRUE;
				SC_VystupVytah.ResetStep:= TRUE;
				SC_VystupVytah.Step:= 100;
			ELSE
				VystupVytah.STAV.PoINIT := TRUE;
				SC_VystupVytah.ResetStep:= TRUE;
				SC_VystupVytah.Step:= 100;
			END_IF

			//********************************************************Automatický režim****************************************************************************//

		100:
			SC_VystupVytah.StepName:='100 - Automaticky Rezim - cakam na navezenie paletky na vytah zo stopra vystupneho dopravnika';
			SC_VystupVytah.IdleTime.PT:= T#500ms;
			SC_VystupVytah.AlarmTime.PT:= T#5s;

			IF VystupVytah.KoniecCyklu THEN
				SC_VystupVytah.ResetStep:= TRUE;
				SC_VystupVytah.Step:= 0;
			ELSIF SC_StoperVystupDopravnika.Step = 105 AND NOT VystupVytah.IN.PritomnostPaletky_IS26 AND NOT VystupVytah.IN.PrechodDopravnikaVytahu_OS6 AND Safety.STAV.BarieraVystupVytahu_AKTIVNA THEN
				SC_VystupVytah.ResetStep:= TRUE;
				SC_VystupVytah.Step:= 105;
			ELSIF VystupVytah.IN.PritomnostPaletky_IS26 AND Safety.STAV.BarieraVystupVytahu_AKTIVNA THEN
				SC_VystupVytah.ResetStep:= TRUE;
				SC_VystupVytah.Step:= 108;
			END_IF

		105:
			SC_VystupVytah.StepName:='105 - Automaticky Rezim - navazam paletku na dopravnik vytahu';
			SC_VystupVytah.IdleTime.PT:= T#200ms;
			SC_VystupVytah.AlarmTime.PT:= T#20s;

			SC_VystupVytah.IdleTime.IN:= VystupVytah.IN.PritomnostPaletky_IS26;

			IF NOT SC_VystupVytah.Switch1 THEN
				VystupVytah.OUT.Dopravnik_ChodVPRED_ELR6:= TRUE;
				SC_VystupVytah.AlarmTime.IN:= TRUE;
				SC_VystupVytah.Switch1:= TRUE;
			END_IF

			IF SC_VystupVytah.IdleTime.Q AND NOT VystupVytah.IN.PrechodDopravnikaVytahu_OS6 THEN
				VystupVytah.OUT.Dopravnik_ChodVPRED_ELR6:= FALSE;
				SC_VystupVytah.ResetStep:= TRUE;
				SC_VystupVytah.Step:= 108;
			ELSIF SC_VystupVytah.AlarmTime.Q THEN
				Alarmy[52]:= TRUE;
				PoruchaVystupnehoVytahu:= TRUE;
				SC_VystupVytah.ResetStep:= TRUE;
				SC_VystupVytah.Step:= 0;
			END_IF

		108:
			SC_VystupVytah.StepName:='108 - Automaticky Rezim - citam cislo paletky';
			SC_VystupVytah.IdleTime.PT:= T#200ms;
			SC_VystupVytah.AlarmTime.PT:= T#10s;

			SC_VystupVytah.IdleTime.IN:= RFID_Hlava_3.STAV.PritomnostCipu;

			IF SC_VystupVytah.IdleTime.Q THEN
				IF RFID_Hlava_3.PAR.PrecitaneCisloPaletky <> '' THEN
					i:=  STRING_TO_USINT(RFID_Hlava_3.PAR.PrecitaneCisloPaletky);
					SC_VystupVytah.ResetStep:= TRUE;
					SC_VystupVytah.Step:= 110;
				ELSE
					Alarmy[62]:= TRUE;
					PoruchaVystupnehoVytahu:= TRUE;
					SC_VystupVytah.ResetStep:= TRUE;
					SC_VystupVytah.Step:= 0;
				END_IF
			END_IF

		110:
			SC_VystupVytah.StepName:='110 - Automaticky Rezim - kontrola stavu paletky';
			SC_VystupVytah.IdleTime.PT:= T#200ms;
			SC_VystupVytah.AlarmTime.PT:= T#10s;

			IF Paletka[i].StavPaletky = 'OK' THEN
				SC_VystupVytah.ResetStep:= TRUE;
				SC_VystupVytah.Step:= 120;
			ELSIF Paletka[i].StavPaletky = 'NG' THEN
				SC_VystupVytah.ResetStep:= TRUE;
				SC_VystupVytah.Step:= 125;
			ELSIF Paletka[i].StavPaletky = 'PR' THEN
				SC_VystupVytah.ResetStep:= TRUE;
				SC_VystupVytah.Step:= 125;
			ELSE
				SC_VystupVytah.ResetStep:= TRUE;
				SC_VystupVytah.Step:= 125;
			END_IF

		120:
			SC_VystupVytah.StepName:='120 - Automaticky Rezim - cakam na odobratie OK kusu a potvrdenie bannerom alebo aktivnou barierou';
			SC_VystupVytah.IdleTime.PT:= T#2s;
			SC_VystupVytah.AlarmTime.PT:= T#10s;

			SC_VystupVytah.IdleTime.IN:= VystupVytah.IN.PritomnostPaletky_IS26 AND Safety.STAV.BarieraVystupVytahu_AKTIVNA;

			VystupVytah.OUT.Banner_ZelenaLED_IOS2:= TRUE;
			VystupVytah.OUT.Banner_CervenaLED_IOS2:= FALSE;

			IF VystupVytah.KoniecCyklu THEN
				SC_VystupVytah.ResetStep:= TRUE;
				SC_VystupVytah.Step:= 0;
			ELSIF VystupVytah.IN.PritomnostPaletky_IS26 AND (NOT VystupVytah.IN.PritomnostProduktu_OS5 OR (Linka.Rezim_Testovania AND SC_VystupVytah.IdleTime.Q)) AND Safety.STAV.BarieraVystupVytahu_AKTIVNA AND VystupVytah.IN.BannerPotvrdeny_IOS2 AND VratnyDopravnik.STAV.PoINIT THEN
				VystupVytah.OUT.Banner_ZelenaLED_IOS2:= FALSE;
				VystupVytah.OUT.Banner_CervenaLED_IOS2:= FALSE;
				SC_VystupVytah.ResetStep:= TRUE;
				SC_VystupVytah.Step:= 130;
			ELSIF VystupVytah.IN.PritomnostPaletky_IS26 AND (NOT VystupVytah.IN.PritomnostProduktu_OS5 OR (Linka.Rezim_Testovania AND SC_VystupVytah.IdleTime.Q)) AND SC_VystupVytah.IdleTime.Q AND NOT VystupVytah_Banner_AKTIVNY AND VratnyDopravnik.STAV.PoINIT THEN
				VystupVytah.OUT.Banner_ZelenaLED_IOS2:= FALSE;
				VystupVytah.OUT.Banner_CervenaLED_IOS2:= FALSE;
				SC_VystupVytah.ResetStep:= TRUE;
				SC_VystupVytah.Step:= 130;
			ELSIF NOT VystupVytah.IN.PritomnostPaletky_IS26 AND Safety.STAV.BarieraVystupVytahu_AKTIVNA THEN
				VystupVytah.OUT.Banner_ZelenaLED_IOS2:= FALSE;
				VystupVytah.OUT.Banner_CervenaLED_IOS2:= FALSE;
				SC_VystupVytah.ResetStep:= TRUE;
				SC_VystupVytah.Step:= 121;
			END_IF

		121:
			SC_VystupVytah.StepName:='121 - Automaticky Rezim - kontrola pritomnosti paletky na dopravniku vytahu';
			SC_VystupVytah.IdleTime.PT:= T#5s;
			SC_VystupVytah.AlarmTime.PT:= T#10s;

			IF NOT SC_VystupVytah.Switch1 THEN
				VystupVytah.OUT.Dopravnik_ChodVPRED_ELR6:= TRUE;
				SC_VystupVytah.IdleTime.IN:= TRUE;
				SC_VystupVytah.Switch1:= TRUE;
			END_IF

			IF VystupVytah.IN.PritomnostPaletky_IS26 THEN
				VystupVytah.OUT.Dopravnik_ChodVPRED_ELR6:= FALSE;
				SC_VystupVytah.ResetStep:= TRUE;
				SC_VystupVytah.Step:= 120;
			ELSIF SC_VystupVytah.IdleTime.Q THEN
				VystupVytah.OUT.Dopravnik_ChodVPRED_ELR6:= FALSE;
				SC_VystupVytah.ResetStep:= TRUE;
				SC_VystupVytah.Step:= 100;
			END_IF

		125:
			SC_VystupVytah.StepName:='125 - Automaticky Rezim - cakam na potvrdenie NG kusu bannerom alebo aktivnou barierou';
			SC_VystupVytah.IdleTime.PT:= T#2s;
			SC_VystupVytah.AlarmTime.PT:= T#10s;

			IF VystupVytah.IN.PritomnostProduktu_OS5 THEN
				VystupVytah.OUT.Banner_ZelenaLED_IOS2:= TRUE;
				VystupVytah.OUT.Banner_CervenaLED_IOS2:= TRUE;
			ELSE
				VystupVytah.OUT.Banner_ZelenaLED_IOS2:= TRUE;
				VystupVytah.OUT.Banner_CervenaLED_IOS2:= FALSE;
			END_IF

			SC_VystupVytah.IdleTime.IN:= VystupVytah.IN.PritomnostPaletky_IS26 AND Safety.STAV.BarieraVystupVytahu_AKTIVNA AND NOT VystupVytah_BannerNG_AKTIVNY AND VratnyDopravnik.STAV.PoINIT;

			IF VystupVytah.KoniecCyklu THEN
				SC_VystupVytah.ResetStep:= TRUE;
				SC_VystupVytah.Step:= 0;
			ELSIF VystupVytah.IN.PritomnostPaletky_IS26 AND Safety.STAV.BarieraVystupVytahu_AKTIVNA AND VystupVytah.IN.BannerPotvrdeny_IOS2 AND VratnyDopravnik.STAV.PoINIT THEN
				VystupVytah.OUT.Banner_ZelenaLED_IOS2:= FALSE;
				VystupVytah.OUT.Banner_CervenaLED_IOS2:= FALSE;
				SC_VystupVytah.ResetStep:= TRUE;
				SC_VystupVytah.Step:= 130;
			ELSIF SC_VystupVytah.IdleTime.Q THEN
				VystupVytah.OUT.Banner_ZelenaLED_IOS2:= FALSE;
				VystupVytah.OUT.Banner_CervenaLED_IOS2:= FALSE;
				SC_VystupVytah.ResetStep:= TRUE;
				SC_VystupVytah.Step:= 130;
			ELSIF NOT VystupVytah.IN.PritomnostPaletky_IS26 AND Safety.STAV.BarieraVystupVytahu_AKTIVNA THEN
				VystupVytah.OUT.Banner_ZelenaLED_IOS2:= FALSE;
				VystupVytah.OUT.Banner_CervenaLED_IOS2:= FALSE;
				SC_VystupVytah.ResetStep:= TRUE;
				SC_VystupVytah.Step:= 128;
			END_IF

		128:
			SC_VystupVytah.StepName:='128 - Automaticky Rezim - kontrola pritomnosti paletky na dopravniku vytahu';
			SC_VystupVytah.IdleTime.PT:= T#2s;
			SC_VystupVytah.AlarmTime.PT:= T#10s;

			IF NOT SC_VystupVytah.Switch1 THEN
				VystupVytah.OUT.Dopravnik_ChodVPRED_ELR6:= TRUE;
				SC_VystupVytah.IdleTime.IN:= TRUE;
				SC_VystupVytah.Switch1:= TRUE;
			END_IF

			IF VystupVytah.IN.PritomnostPaletky_IS26 THEN
				VystupVytah.OUT.Dopravnik_ChodVPRED_ELR6:= FALSE;
				SC_VystupVytah.ResetStep:= TRUE;
				SC_VystupVytah.Step:= 125;
			ELSIF SC_VystupVytah.IdleTime.Q THEN
				VystupVytah.OUT.Dopravnik_ChodVPRED_ELR6:= FALSE;
				SC_VystupVytah.ResetStep:= TRUE;
				SC_VystupVytah.Step:= 100;
			END_IF

		130:
			SC_VystupVytah.StepName:='130 - Automaticky Rezim - presuvam vytah do spodnej pozicie vyvazania';
			SC_VystupVytah.IdleTime.PT:= T#3s;
			SC_VystupVytah.AlarmTime.PT:= T#5s;

			VystupVytah.OUT.Banner_CervenaLED_IOS2:= TRUE;
			VystupVytah.PAR.Zdvih_ZadanaRychlost:= 50;
			VystupVytah.PAR.Zdvih_ZadanaPozicia:= RemPremenne.VystupVytah_PozVyvazania;

			IF NOT SC_VystupVytah.Switch1 AND SC_OvlMenica.Step = 1 THEN
				Zdvih_POLOHUJ:= TRUE;
				VystupVytah.OUT.Dopravnik_ChodVPRED_ELR6:= TRUE;
				VystupnyVytah_Statistika.IN.START_MeraniaCasu:= TRUE;
				VystupnyVytah_Statistika.IN.ZAPIS_MeraniaCasu:= TRUE;
				SC_VystupVytah.Switch1:= TRUE;
			END_IF

			IF VystupVytah.STAV.VytahNapolohovany THEN
				VystupVytah.STAV.VytahNapolohovany:= FALSE;
				VystupVytah.OUT.Dopravnik_ChodVPRED_ELR6:= FALSE;
				SC_VystupVytah.ResetStep:= TRUE;
				SC_VystupVytah.Step:= 135;
			ELSIF NOT Safety.STAV.BarieraVystupVytahu_AKTIVNA THEN
				Alarmy[50]:= TRUE;
				PoruchaVystupnehoVytahu:= TRUE;
				SC_VystupVytah.ResetStep:= TRUE;
				SC_VystupVytah.Step:= 0;
			ELSIF VystupVytah.IN.PrechodDopravnikaVytahu_OS6 THEN
				Alarmy[51]:= TRUE;
				PoruchaVystupnehoVytahu:= TRUE;
				SC_VystupVytah.ResetStep:= TRUE;
				SC_VystupVytah.Step:= 0;
			END_IF

		135:
			SC_VystupVytah.StepName:='135 - Automaticky Rezim - vyvezenie paletky na vratny dopravnik';
			SC_VystupVytah.IdleTime.PT:= T#200ms;
			SC_VystupVytah.AlarmTime.PT:= T#2s;

			IF NOT SC_VystupVytah.Switch1 THEN
				VystupVytah.OUT.Dopravnik_ChodVZAD_ELR6:= TRUE;
				SC_VystupVytah.Switch1:= TRUE;
			END_IF

			IF EDGENEG(VystupVytah.IN.PrechodDopravnikaVytahu_OS6) THEN
				SC_VystupVytah.IdleTime.IN:= TRUE;
			END_IF

			IF SC_VystupVytah.IdleTime.Q AND NOT VystupVytah.IN.PritomnostPaletky_IS26 AND NOT VystupVytah.IN.PrechodDopravnikaVytahu_OS6 THEN
				VystupVytah.OUT.Dopravnik_ChodVZAD_ELR6:= FALSE;
				SC_VystupVytah.ResetStep:= TRUE;
				SC_VystupVytah.Step:= 140;
			END_IF

		140:
			SC_VystupVytah.StepName:='140 - Automaticky Rezim - cakam na presun vytahu do hornej pozicie navazania';
			SC_VystupVytah.IdleTime.PT:= T#1s;
			SC_VystupVytah.AlarmTime.PT:= T#10s;

			SC_VystupVytah.IdleTime.IN:= Safety.STAV.BarieraVystupVytahu_AKTIVNA AND NOT VystupVytah.IN.PrechodDopravnikaVytahu_OS6;

			IF SC_VystupVytah.IdleTime.Q THEN
				SC_VystupVytah.ResetStep:= TRUE;
				SC_VystupVytah.Step:= 143;
			END_IF

		143:
			SC_VystupVytah.StepName:='143 - Automaticky Rezim - presuvam vytah do hornej pozicie navazania';
			SC_VystupVytah.IdleTime.PT:= T#500ms;
			SC_VystupVytah.AlarmTime.PT:= T#10s;

			VystupVytah.OUT.Banner_CervenaLED_IOS2:= TRUE;
			VystupVytah.PAR.Zdvih_ZadanaRychlost:= 50;
			VystupVytah.PAR.Zdvih_ZadanaPozicia:= RemPremenne.VystupVytah_PozNavazania;

			IF NOT SC_VystupVytah.Switch1 AND SC_OvlMenica.Step = 1 THEN
				Zdvih_POLOHUJ:= TRUE;
				SC_VystupVytah.Switch1:= TRUE;
			END_IF

			IF VystupVytah.STAV.VytahNapolohovany THEN
				VystupVytah.STAV.VytahNapolohovany:= FALSE;
				VystupVytah.OUT.Banner_CervenaLED_IOS2:= FALSE;
				SC_VystupVytah.ResetStep:= TRUE;
				SC_VystupVytah.Step:= 100;
			ELSIF NOT Safety.STAV.BarieraVystupVytahu_AKTIVNA THEN
				Alarmy[50]:= TRUE;
				PoruchaVystupnehoVytahu:= TRUE;
				SC_VystupVytah.ResetStep:= TRUE;
				SC_VystupVytah.Step:= 0;
			ELSIF VystupVytah.IN.PrechodDopravnikaVytahu_OS6 THEN
				Alarmy[51]:= TRUE;
				PoruchaVystupnehoVytahu:= TRUE;
				SC_VystupVytah.ResetStep:= TRUE;
				SC_VystupVytah.Step:= 0;
			END_IF

			//*******************************************************Manuálny režim*******************************************************************************//
		700:
			SC_VystupVytah.StepName:='700 - Manualny Rezim';
			SC_VystupVytah.IdleTime.PT:= T#8s;
			SC_VystupVytah.AlarmTime.PT:= T#5s;

			//Ovládanie dopravníka//
			IF VystupVytah.RR_Dopravnik_VPRED THEN
				VystupVytah.OUT.Dopravnik_ChodVZAD_ELR6:= FALSE;
				VystupVytah.OUT.Dopravnik_ChodVPRED_ELR6:= TRUE;
			ELSIF VystupVytah.RR_Dopravnik_VZAD THEN
				VystupVytah.OUT.Dopravnik_ChodVPRED_ELR6:= FALSE;
				VystupVytah.OUT.Dopravnik_ChodVZAD_ELR6:= TRUE;
			ELSE
				VystupVytah.OUT.Dopravnik_ChodVPRED_ELR6:= FALSE;
				VystupVytah.OUT.Dopravnik_ChodVZAD_ELR6:= FALSE;
			END_IF

	END_CASE

END_PROGRAM

PROGRAM _EXIT
	(* Insert code here *)

END_PROGRAM
```

#### Variables.var - Local variables
```iecst
VAR
	SC_OvlMenica : SequenceControlTyp := (0);
	Zdvih_JoggHORE : BOOL := FALSE;
	Zdvih_JoggDOLE : BOOL := FALSE;
	Zdvih_POLOHUJ : BOOL := FALSE;
	Zdvih_HOME : BOOL := FALSE;
	VstupnePoleUSINT : ARRAY[1..20] OF USINT;
	VystupnePoleStringov : ARRAY[1..20] OF STRING[80];
	h : USINT := 0;
	PocetZnakovUDINT : UDINT;
	PocetZnakovUSINT : USINT;
	g : USINT := 0;
	AktualNacitanyZnak : USINT;
	i : USINT := 0;
END_VAR
```

#### OvlMenica.st
```iecst
ACTION OvlMenica:

	//Otáčka motora = zdvih 10 mm//

	//CANopen adresa meniča - 36//

	//Volanie funkčného bloku//
	VystupVytah.MenicZdvihu_FM3();

	//Volanie funkcie SequenceControl//
	SequenceControl(SC:= SC_OvlMenica);

	//Prepnutie meniča do stavu READY//
	IF EDGEPOS(Safety.STAV.SafetyPLC_Nabehlo)THEN
		IF NOT VystupVytah.MenicZdvihu_FM3.STAV.READY THEN
			VystupVytah.MenicZdvihu_FM3.CMD.Potvrd_PORUCHU:= TRUE;
		END_IF
	ELSIF EDGEPOS(Safety.STAV.ZonaVystupnyVytah_AKTIVNA)THEN
		IF NOT VystupVytah.MenicZdvihu_FM3.STAV.READY THEN
			VystupVytah.MenicZdvihu_FM3.CMD.Potvrd_PORUCHU:= TRUE;
		END_IF
	END_IF

	//Parametre meniča//
	VystupVytah.MenicZdvihu_FM3.PAR.TypKomunikacieProfinet:= 0;
	VystupVytah.MenicZdvihu_FM3.PAR.ZadanaPozicia_MM:= (VystupVytah.PAR.Zdvih_ZadanaPozicia * 100);
	VystupVytah.STAV.Zdvih_AktualnaPozicia:= (VystupVytah.MenicZdvihu_FM3.PAR.AktualnaPozicia_MM/100);
	VystupVytah.STAV.Zdvih_AktualnaRychlost:= VystupVytah.MenicZdvihu_FM3.PAR.AktualnaFrekvencia_Hz;
	VystupVytah.STAV.Zdvih_HomingOK:= VystupVytah.MenicZdvihu_FM3.STAV.Homing_OK;
	VystupVytah.STAV.Zdvih_PoziciaDosiahnuta:= VystupVytah.MenicZdvihu_FM3.STAV.Pozicia_DOSIAHNUTA;
	VystupVytah.STAV.Zdvih_BUSY:= VystupVytah.MenicZdvihu_FM3.STAV.RUN;

	//Preposielanie IO meniča cez komunikáciu//
	VystupVytah.IN.ReferencnySnimacZdvihu:= VystupVytah.MenicZdvihu_FM3.PAR.BUS_OUT_Bit_0;
	VystupVytah.IN.HornyLimitZdvihu:= VystupVytah.MenicZdvihu_FM3.PAR.BUS_OUT_Bit_1;
	VystupVytah.MenicZdvihu_FM3.PAR.BUS_IN_Bit_0:= VystupVytah.IN.SpodnyLimitZdvihu;

	IF Zdvih_HOME THEN
		VystupVytah.IN.SpodnyLimitZdvihu:= TRUE;
	ELSE
		VystupVytah.IN.SpodnyLimitZdvihu:= NOT VystupVytah.IN.ReferencnySnimacZdvihu;
	END_IF

	IF NOT Safety.STAV.ZonaVystupnyVytah_AKTIVNA THEN
		SC_OvlMenica.Step:= 0;
	END_IF

	CASE SC_OvlMenica.Step OF

		0:
			SC_OvlMenica.StepName:= '0 - Nulovanie';
			Zdvih_JoggHORE:= FALSE;
			Zdvih_JoggDOLE:= FALSE;
			Zdvih_POLOHUJ:= FALSE;
			Zdvih_HOME:= FALSE;
			VystupVytah.MenicZdvihu_FM3.CMD.HOME:= FALSE;
			VystupVytah.MenicZdvihu_FM3.CMD.Chod_VPRED:= FALSE;
			VystupVytah.MenicZdvihu_FM3.CMD.Chod_VZAD:= FALSE;
			VystupVytah.MenicZdvihu_FM3.CMD.Polohuj:= FALSE;
			VystupVytah.STAV.Homing_BUSY:= FALSE;

			IF SC_VystupVytah.Step <> 0 AND VystupVytah.MenicZdvihu_FM3.STAV.READY AND NOT VystupVytah.MenicZdvihu_FM3.STAV.PORUCHA AND Safety.STAV.ZonaVystupnyVytah_AKTIVNA THEN
				SC_OvlMenica.ResetStep:= TRUE;
				SC_OvlMenica.Step:= 1;
			END_IF

		1:
			SC_OvlMenica.StepName:= '1 - Rozhodnutie o cinnosti';
			IF Zdvih_JoggHORE THEN
				SC_OvlMenica.Step:= 10;
			ELSIF Zdvih_JoggDOLE THEN
				SC_OvlMenica.Step:= 20;
			ELSIF Zdvih_HOME THEN
				SC_OvlMenica.Step:= 30;
			ELSIF Zdvih_POLOHUJ THEN
				SC_OvlMenica.Step:= 40;
			END_IF

		10:
			SC_OvlMenica.StepName:= '10 - Jogg HORE';
			SC_OvlMenica.IdleTime.PT:= T#3s;
			SC_OvlMenica.AlarmTime.PT:= T#3s;

			VystupVytah.MenicZdvihu_FM3.PAR.ZadanaFrekvencia_Hz:= VystupVytah.PAR.Zdvih_ZadanaJoggRychlost;

			IF NOT SC_OvlMenica.Switch1 AND VystupVytah.IN.HornyLimitZdvihu THEN
				VystupVytah.MenicZdvihu_FM3.CMD.Chod_VPRED:= TRUE;
				SC_OvlMenica.Switch1:= TRUE;
			END_IF

			IF NOT Zdvih_JoggHORE THEN
				SC_OvlMenica.ResetStep:= TRUE;
				SC_OvlMenica.Step:= 0;
			ELSIF NOT VystupVytah.IN.HornyLimitZdvihu THEN
				SC_OvlMenica.ResetStep:= TRUE;
				SC_OvlMenica.Step:= 0;
			END_IF

		20:
			SC_OvlMenica.StepName:= '20 - Jogg DOLE';
			SC_OvlMenica.IdleTime.PT:= T#3s;
			SC_OvlMenica.AlarmTime.PT:= T#3s;

			VystupVytah.MenicZdvihu_FM3.PAR.ZadanaFrekvencia_Hz:= VystupVytah.PAR.Zdvih_ZadanaJoggRychlost;

			IF NOT SC_OvlMenica.Switch1 AND VystupVytah.IN.SpodnyLimitZdvihu THEN
				VystupVytah.MenicZdvihu_FM3.CMD.Chod_VZAD:= TRUE;
				SC_OvlMenica.Switch1:= TRUE;
			END_IF

			IF NOT Zdvih_JoggDOLE THEN
				SC_OvlMenica.ResetStep:= TRUE;
				SC_OvlMenica.Step:= 0;
			ELSIF NOT VystupVytah.IN.SpodnyLimitZdvihu THEN
				SC_OvlMenica.ResetStep:= TRUE;
				SC_OvlMenica.Step:= 0;
			END_IF

		30:
			SC_OvlMenica.StepName:= '30 - Homing - kontrola referencneho snimaca';
			SC_OvlMenica.IdleTime.PT:= T#500ms;
			SC_OvlMenica.AlarmTime.PT:= T#3s;

			VystupVytah.STAV.Homing_BUSY:= TRUE;

			IF VystupVytah.IN.ReferencnySnimacZdvihu THEN
				SC_OvlMenica.ResetStep:= TRUE;
				SC_OvlMenica.Step:= 31;
			ELSE
				SC_OvlMenica.ResetStep:= TRUE;
				SC_OvlMenica.Step:= 32;
			END_IF

		31:
			SC_OvlMenica.StepName:= '31 - Homing - presun vytahu nad referencny snimac';
			SC_OvlMenica.IdleTime.PT:= T#1s;
			SC_OvlMenica.AlarmTime.PT:= T#2s;

			SC_OvlMenica.IdleTime.IN:= NOT VystupVytah.IN.ReferencnySnimacZdvihu;

			IF NOT SC_OvlMenica.Switch1 THEN
				VystupVytah.MenicZdvihu_FM3.CMD.Chod_VPRED:= TRUE;
				SC_OvlMenica.Switch1:= TRUE;
			END_IF

			IF SC_OvlMenica.IdleTime.Q THEN
				VystupVytah.MenicZdvihu_FM3.CMD.Chod_VPRED:= FALSE;
				SC_OvlMenica.AlarmTime.IN:= TRUE;
			END_IF

			IF SC_OvlMenica.AlarmTime.Q THEN
				SC_OvlMenica.ResetStep:= TRUE;
				SC_OvlMenica.Step:= 32;
			END_IF

		32:
			SC_OvlMenica.StepName:= '32 - Homing - spustenie homingu';
			SC_OvlMenica.IdleTime.PT:= T#500ms;
			SC_OvlMenica.AlarmTime.PT:= T#3s;

			IF NOT SC_OvlMenica.Switch1 THEN
				VystupVytah.MenicZdvihu_FM3.CMD.HOME:= TRUE;
				SC_OvlMenica.IdleTime.IN:= TRUE;
				SC_OvlMenica.Switch1:= TRUE;
			END_IF

			IF VystupVytah.STAV.Zdvih_HomingOK AND SC_OvlMenica.IdleTime.Q THEN
				SC_OvlMenica.ResetStep:= TRUE;
				SC_OvlMenica.Step:= 0;
			ELSIF NOT Zdvih_HOME THEN
				SC_OvlMenica.ResetStep:= TRUE;
				SC_OvlMenica.Step:= 0;
			END_IF

		40:
			SC_OvlMenica.StepName:= '40 - Polohovanie';
			SC_OvlMenica.IdleTime.PT:= T#1s;
			SC_OvlMenica.AlarmTime.PT:= T#3s;

			VystupVytah.MenicZdvihu_FM3.PAR.ZadanaFrekvencia_Hz:= VystupVytah.PAR.Zdvih_ZadanaRychlost;

			IF NOT SC_OvlMenica.Switch1 THEN
				VystupVytah.MenicZdvihu_FM3.CMD.Polohuj:= TRUE;
				SC_OvlMenica.IdleTime.IN:= TRUE;
				SC_OvlMenica.Switch1:= TRUE;
			END_IF

			IF (*(VystupVytah.STAV.Zdvih_AktualnaPozicia = VystupVytah.PAR.Zdvih_ZadanaPozicia) AND*) SC_OvlMenica.IdleTime.Q AND VystupVytah.STAV.Zdvih_PoziciaDosiahnuta THEN
				VystupVytah.STAV.VytahNapolohovany:= TRUE;
				SC_OvlMenica.ResetStep:= TRUE;
				SC_OvlMenica.Step:= 0;
			ELSIF NOT Zdvih_POLOHUJ THEN
				SC_OvlMenica.ResetStep:= TRUE;
				SC_OvlMenica.Step:= 0;
			END_IF

	END_CASE

END_ACTION
```

#### OvlCitackyRFID.st
```iecst
ACTION OvlCitackyRFID:

		//***********************************************************************Riadenie RFID hlavy 3 - Pozícia dopravníka NG**********************************************************************//

	//Volanie funkcie SequenceControl//
	SequenceControl(SC:= SC_Hlava_3);

	//*************************Komunikácia*******************************//
	//INPUTS//
	RFID_Hlava_3.STAV.PritomnostCipu:= RFID_Hlava_3.IN.BYTE_IN[0].0;
	RFID_Hlava_3.IN.Bit_CP:= RFID_Hlava_3.IN.BYTE_IN[0].0;
	RFID_Hlava_3.IN.Bit_AA:= RFID_Hlava_3.IN.BYTE_IN[0].1;
	RFID_Hlava_3.IN.Bit_AE:= RFID_Hlava_3.IN.BYTE_IN[0].2;
	RFID_Hlava_3.IN.Bit_AF:= RFID_Hlava_3.IN.BYTE_IN[0].3;
	RFID_Hlava_3.IN.Bit_MT:= RFID_Hlava_3.IN.BYTE_IN[0].4;
	RFID_Hlava_3.IN.Bit_TO:= RFID_Hlava_3.IN.BYTE_IN[0].5;
	RFID_Hlava_3.IN.Bit_HF:= RFID_Hlava_3.IN.BYTE_IN[0].6;
	RFID_Hlava_3.IN.Bit_BB:= RFID_Hlava_3.IN.BYTE_IN[0].7;

	//OUTPUTS//
	RFID_Hlava_3.OUT.BYTE_OUT[0].0:= RFID_Hlava_3.OUT.Bit_AV;
	RFID_Hlava_3.OUT.BYTE_OUT[31].0:= RFID_Hlava_3.OUT.Bit_AV;
	RFID_Hlava_3.OUT.BYTE_OUT[0].2:= RFID_Hlava_3.OUT.Bit_GR;
	RFID_Hlava_3.OUT.BYTE_OUT[31].2:= RFID_Hlava_3.OUT.Bit_GR;
	RFID_Hlava_3.OUT.BYTE_OUT[0].5:= RFID_Hlava_3.OUT.Bit_KA;
	RFID_Hlava_3.OUT.BYTE_OUT[31].5:= RFID_Hlava_3.OUT.Bit_KA;
	RFID_Hlava_3.OUT.BYTE_OUT[0].6:= RFID_Hlava_3.OUT.Bit_TI;
	RFID_Hlava_3.OUT.BYTE_OUT[31].6:= RFID_Hlava_3.OUT.Bit_TI;

	//Prečítané znaky//
	RFID_Hlava_3.PAR.PrecitaneCisloPaletky_POLE[0]:= RFID_Hlava_3.IN.BYTE_IN[1];
	RFID_Hlava_3.PAR.PrecitaneCisloPaletky_POLE[1]:= RFID_Hlava_3.IN.BYTE_IN[2];
	RFID_Hlava_3.PAR.PrecitaneCisloPaletky_POLE[2]:= RFID_Hlava_3.IN.BYTE_IN[3];
	RFID_Hlava_3.PAR.PrecitaneCisloPaletky_POLE[3]:= RFID_Hlava_3.IN.BYTE_IN[4];
	RFID_Hlava_3.PAR.PrecitaneCisloPaletky_POLE[4]:= RFID_Hlava_3.IN.BYTE_IN[5];
	RFID_Hlava_3.PAR.PrecitaneCisloPaletky_POLE[5]:= RFID_Hlava_3.IN.BYTE_IN[6];
	RFID_Hlava_3.PAR.PrecitaneCisloPaletky_POLE[6]:= RFID_Hlava_3.IN.BYTE_IN[7];
	RFID_Hlava_3.PAR.PrecitaneCisloPaletky_POLE[7]:= RFID_Hlava_3.IN.BYTE_IN[8];
	RFID_Hlava_3.PAR.PrecitaneCisloPaletky_POLE[8]:= RFID_Hlava_3.IN.BYTE_IN[9];
	RFID_Hlava_3.PAR.PrecitaneCisloPaletky_POLE[9]:= RFID_Hlava_3.IN.BYTE_IN[10];

	brsmemcpy(ADR(RFID_Hlava_3.PAR.Precitane_Cislo_Typ_Paletky),ADR(RFID_Hlava_3.PAR.PrecitaneCisloPaletky_POLE),SIZEOF(RFID_Hlava_3.PAR.PrecitaneCisloPaletky_POLE));

	//Rozdelenie prečítanej správy na číslo paletky a model//
	IF RFID_Hlava_3.STAV.PritomnostCipu THEN
		brsmemset(ADR(VstupnePoleUSINT),0,SIZEOF(VstupnePoleUSINT)); //Vymazanie vstupneho pola
		brsmemset(ADR(VystupnePoleStringov),0,SIZEOF(VystupnePoleStringov)); //Vymazanie výstupneho pola znakov
		PocetZnakovUDINT := brsstrlen(ADR(RFID_Hlava_3.PAR.Precitane_Cislo_Typ_Paletky)); //Zistenie počtu znakov vstupnej spravy
		PocetZnakovUSINT:= UDINT_TO_USINT(PocetZnakovUDINT);
		brsmemcpy(ADR(VstupnePoleUSINT),ADR(RFID_Hlava_3.PAR.Precitane_Cislo_Typ_Paletky),SIZEOF(RFID_Hlava_3.PAR.Precitane_Cislo_Typ_Paletky)); //Vyplnenie polia znakmy vstupnej správy
		h:= 1;
		FOR g:= 1 TO PocetZnakovUSINT BY 1 DO
			IF VstupnePoleUSINT[g] <> 59 THEN //59 je oddelovací znak bodkočiarka
				AktualNacitanyZnak:= VstupnePoleUSINT[g];
				brsstrcat(ADR(VystupnePoleStringov[h]),ADR(AktualNacitanyZnak));
			ELSE
				h:= h + 1;
			END_IF
		END_FOR
		RFID_Hlava_3.PAR.PrecitaneCisloPaletky:= VystupnePoleStringov[1];
		RFID_Hlava_3.PAR.PrecitanyTypPaletky:= VystupnePoleStringov[2];
	ELSE
		RFID_Hlava_3.PAR.PrecitaneCisloPaletky:= '';
		RFID_Hlava_3.PAR.PrecitanyTypPaletky:= '';
	END_IF

	CASE SC_Hlava_3.Step OF

		0:
			SC_Hlava_3.StepName:= '0 - Nulovanie';
			RFID_Hlava_3.CMD.CitajDATA:= FALSE;
			RFID_Hlava_3.CMD.ZapisDATA:= FALSE;
			RFID_Hlava_3.CMD.CitaciuHlavu_VYPNI:= FALSE;
			RFID_Hlava_3.OUT.Bit_AV:= FALSE;
			RFID_Hlava_3.OUT.Bit_GR:= FALSE;
			RFID_Hlava_3.OUT.Bit_TI:= FALSE;
			RFID_Hlava_3.OUT.Bit_KA:= FALSE;

			IF RFID_Hlava_3.STAV.PritomnostCipu THEN
				SC_Hlava_3.ResetStep:= TRUE;
				SC_Hlava_3.Step:= 1;
			END_IF

		1:
			SC_Hlava_3.StepName:= '1 - Rozhodnutie o cinnosti';
			IF NOT RFID_Hlava_3.STAV.PritomnostCipu THEN
				SC_Hlava_3.Step:= 0;
			ELSIF RFID_Hlava_3.CMD.CitajDATA THEN
				RFID_Hlava_3.STAV.CitanieDat_OK:= FALSE;
				RFID_Hlava_3.STAV.CitanieDat_ERROR:= FALSE;
				SC_Hlava_3.Step:= 10;
			ELSIF RFID_Hlava_3.CMD.ZapisDATA THEN
				RFID_Hlava_3.STAV.ZapisDat_OK:= FALSE;
				RFID_Hlava_3.STAV.ZapisDat_ERROR:= FALSE;
				SC_Hlava_3.Step:= 20;
			ELSIF RFID_Hlava_3.CMD.CitaciuHlavu_VYPNI THEN
				SC_Hlava_3.Step:= 30;
			END_IF

		10:
			SC_Hlava_3.StepName:= '10 - Citanie dat';
			SC_Hlava_3.IdleTime.PT:= T#3s;
			SC_Hlava_3.AlarmTime.PT:= T#6s;

			RFID_Hlava_3.IN.Old_Bit_TO:= RFID_Hlava_3.IN.Bit_TO;
			RFID_Hlava_3.OUT.BYTE_OUT[1]:= 1; //Kommand - 1 - čítanie, 2 - zápis
			RFID_Hlava_3.OUT.BYTE_OUT[2]:= 0; //Štartovacia adresa čítania (LSB) - na 2 byte začína zapisovať načítané znaky
			RFID_Hlava_3.OUT.BYTE_OUT[3]:= 0; //Štartovacia adresa čítania (HSB)
			RFID_Hlava_3.OUT.BYTE_OUT[4]:= 10; //Počet bajtov čítania (LSB) - 10 znakov
			RFID_Hlava_3.OUT.BYTE_OUT[5]:= 0; //Počet bajtov čítania (HSB)
			RFID_Hlava_3.OUT.Bit_AV:= TRUE;

			SC_Hlava_3.ResetStep:= TRUE;
			SC_Hlava_3.Step:= 11;

		11:
			SC_Hlava_3.StepName:= '11 - Citanie dat';
			SC_Hlava_3.IdleTime.PT:= T#3s;
			SC_Hlava_3.AlarmTime.PT:= T#2s;

			IF RFID_Hlava_3.IN.Bit_AA AND RFID_Hlava_3.IN.Bit_AE AND (RFID_Hlava_3.IN.Old_Bit_TO <> RFID_Hlava_3.IN.Bit_TO) THEN
				RFID_Hlava_3.STAV.CitanieDat_OK:= TRUE;
				SC_Hlava_3.ResetStep:= TRUE;
				SC_Hlava_3.Step:= 12;
			ELSIF RFID_Hlava_3.IN.Bit_AF THEN
				RFID_Hlava_3.STAV.CitanieDat_ERROR:= TRUE;
				SC_Hlava_3.ResetStep:= TRUE;
				SC_Hlava_3.Step:= 12;
			END_IF

		12:
			SC_Hlava_3.StepName:= '12 - Citanie dat';
			SC_Hlava_3.IdleTime.PT:= T#3s;
			SC_Hlava_3.AlarmTime.PT:= T#6s;

			RFID_Hlava_3.OUT.Bit_AV:= FALSE;

			IF NOT RFID_Hlava_3.IN.Bit_AA AND NOT RFID_Hlava_3.IN.Bit_AE AND NOT RFID_Hlava_3.IN.Bit_AF THEN
				SC_Hlava_3.ResetStep:= TRUE;
				SC_Hlava_3.Step:= 0;
			END_IF

		20:
			SC_Hlava_3.StepName:= '20 - Zápis dat';
			SC_Hlava_3.IdleTime.PT:= T#3s;
			SC_Hlava_3.AlarmTime.PT:= T#6s;

			RFID_Hlava_3.IN.Old_Bit_TO:= RFID_Hlava_3.IN.Bit_TO;
			RFID_Hlava_3.OUT.BYTE_OUT[1]:= 2; //Kommand - 1 - čítanie, 2 - zápis
			RFID_Hlava_3.OUT.BYTE_OUT[2]:= 0; //Štartovacia adresa zápisu (LSB) - na 2 byte začína zapisovať znaky
			RFID_Hlava_3.OUT.BYTE_OUT[3]:= 0; //Štartovacia adresa zápisu (HSB)
			RFID_Hlava_3.OUT.BYTE_OUT[4]:= 10; //Počet bajtov zápisu (LSB) - 10 znakov
			RFID_Hlava_3.OUT.BYTE_OUT[5]:= 0; //Počet bajtov zápisu (HSB)
			RFID_Hlava_3.OUT.Bit_AV:= TRUE;

			SC_Hlava_3.ResetStep:= TRUE;
			SC_Hlava_3.Step:= 21;

		21:
			SC_Hlava_3.StepName:= '21 - Zápis dat';
			SC_Hlava_3.IdleTime.PT:= T#3s;
			SC_Hlava_3.AlarmTime.PT:= T#2s;

			IF RFID_Hlava_3.IN.Bit_AA AND (RFID_Hlava_3.IN.Old_Bit_TO <> RFID_Hlava_3.IN.Bit_TO) THEN
				SC_Hlava_3.ResetStep:= TRUE;
				SC_Hlava_3.Step:= 22;
			END_IF

		22:
			SC_Hlava_3.StepName:= '21 - Zápis dat';
			SC_Hlava_3.IdleTime.PT:= T#3s;
			SC_Hlava_3.AlarmTime.PT:= T#6s;

			brsstrcpy(ADR(RFID_Hlava_3.PAR.ZadaneCisloPaletky_POLE),ADR(RFID_Hlava_3.PAR.Zadane_Cislo_Typ_Paletky));
			RFID_Hlava_3.OUT.BYTE_OUT[1]:= RFID_Hlava_3.PAR.ZadaneCisloPaletky_POLE[0];
			RFID_Hlava_3.OUT.BYTE_OUT[2]:= RFID_Hlava_3.PAR.ZadaneCisloPaletky_POLE[1];
			RFID_Hlava_3.OUT.BYTE_OUT[3]:= RFID_Hlava_3.PAR.ZadaneCisloPaletky_POLE[2];
			RFID_Hlava_3.OUT.BYTE_OUT[4]:= RFID_Hlava_3.PAR.ZadaneCisloPaletky_POLE[3];
			RFID_Hlava_3.OUT.BYTE_OUT[5]:= RFID_Hlava_3.PAR.ZadaneCisloPaletky_POLE[4];
			RFID_Hlava_3.OUT.BYTE_OUT[6]:= RFID_Hlava_3.PAR.ZadaneCisloPaletky_POLE[5];
			RFID_Hlava_3.OUT.BYTE_OUT[7]:= RFID_Hlava_3.PAR.ZadaneCisloPaletky_POLE[6];
			RFID_Hlava_3.OUT.BYTE_OUT[8]:= RFID_Hlava_3.PAR.ZadaneCisloPaletky_POLE[7];
			RFID_Hlava_3.OUT.BYTE_OUT[9]:= RFID_Hlava_3.PAR.ZadaneCisloPaletky_POLE[8];
			RFID_Hlava_3.OUT.BYTE_OUT[10]:= RFID_Hlava_3.PAR.ZadaneCisloPaletky_POLE[9];

			IF RFID_Hlava_3.OUT.Bit_TI THEN
				RFID_Hlava_3.OUT.Bit_TI:= FALSE;
				SC_Hlava_3.ResetStep:= TRUE;
				SC_Hlava_3.Step:= 23;
			ELSE
				RFID_Hlava_3.OUT.Bit_TI:= TRUE;
				SC_Hlava_3.ResetStep:= TRUE;
				SC_Hlava_3.Step:= 23;
			END_IF

		23:
			SC_Hlava_3.StepName:= '23 - Zápis dat';
			SC_Hlava_3.IdleTime.PT:= T#3s;
			SC_Hlava_3.AlarmTime.PT:= T#2s;

			IF RFID_Hlava_3.IN.Bit_AE THEN
				RFID_Hlava_3.STAV.ZapisDat_OK:= TRUE;
				SC_Hlava_3.ResetStep:= TRUE;
				SC_Hlava_3.Step:= 24;
			ELSIF RFID_Hlava_3.IN.Bit_AF THEN
				RFID_Hlava_3.STAV.ZapisDat_ERROR:= TRUE;
				SC_Hlava_3.ResetStep:= TRUE;
				SC_Hlava_3.Step:= 24;
			END_IF

		24:
			SC_Hlava_3.StepName:= '22 - Zápis dat';
			SC_Hlava_3.IdleTime.PT:= T#3s;
			SC_Hlava_3.AlarmTime.PT:= T#6s;

			RFID_Hlava_3.OUT.Bit_AV:= FALSE;

			IF NOT RFID_Hlava_3.IN.Bit_AA AND NOT RFID_Hlava_3.IN.Bit_AE AND NOT RFID_Hlava_3.IN.Bit_AF THEN
				SC_Hlava_3.ResetStep:= TRUE;
				SC_Hlava_3.Step:= 0;
			END_IF

		30:
			SC_Hlava_3.StepName:= '30 - Vypnutie citacej hlavy';
			SC_Hlava_3.IdleTime.PT:= T#3s;
			SC_Hlava_3.AlarmTime.PT:= T#2s;

			RFID_Hlava_3.OUT.Bit_KA:= TRUE;

			IF NOT RFID_Hlava_3.CMD.CitaciuHlavu_VYPNI THEN
				SC_Hlava_3.ResetStep:= TRUE;
				SC_Hlava_3.Step:= 0;
			END_IF

	END_CASE

END_ACTION
```

### Program Logical/Program/StoperVratDopravnika (IEC)

#### Main.st - Init, cyclic, exit code
```iecst
PROGRAM _INIT
	(* Insert code here *)

END_PROGRAM

PROGRAM _CYCLIC

	//Volanie funkcie SequenceControl//
	SequenceControl(SC:= SC_StoperVratDopravnika);

	//Reset sekcie //
	IF StoperVratDopravnika.Reset THEN
		SC_StoperVratDopravnika.Step:= 0;
		StoperVratDopravnika.Reset:= FALSE;
	ELSIF NOT Safety.STAV.ZonaCS_AKTIVNA THEN
		SC_StoperVratDopravnika.Step:= 0;
	END_IF

	CASE SC_StoperVratDopravnika.Step OF

		0:
			SC_StoperVratDopravnika.StepName:='0 - Nulovanie';
			StoperVratDopravnika.Automat:= FALSE;
			StoperVratDopravnika.KoniecCyklu:= FALSE;
			StoperVratDopravnika.Manual:= FALSE;
			StoperVratDopravnika.STAV.PoINIT:= FALSE;
			StoperVratDopravnika.OUT.StoperZASUN_YV012:= FALSE;

			IF Safety.STAV.ZonaCS_AKTIVNA AND Linka.IN.TlakVzduchu_OK_S2 AND NOT NastalaPorucha AND Linka.STAV.Hardware_OK THEN
				SC_StoperVratDopravnika.ResetStep:= TRUE;
				SC_StoperVratDopravnika.Step:= 1;
			END_IF

		1:
			SC_StoperVratDopravnika.StepName:='1 - Cakam na spustenie vyroby';
			StoperVratDopravnika.KoniecCyklu:= FALSE;
			IF StoperVratDopravnika.Automat THEN
				SC_StoperVratDopravnika.Step:= 2;
			ELSIF StoperVratDopravnika.Manual THEN
				SC_StoperVratDopravnika.Step:= 700;
			END_IF

			//********************************************************Inicializácia****************************************************************************//

		2:
			SC_StoperVratDopravnika.StepName:='2 - Inicializacia - cakam na spustenie inicializacie';
			SC_StoperVratDopravnika.IdleTime.PT:= T#4s;
			SC_StoperVratDopravnika.AlarmTime.PT:= T#5s;

			IF VratnyDopravnik.STAV.PoINIT THEN
				SC_StoperVratDopravnika.ResetStep:= TRUE;
				SC_StoperVratDopravnika.Step:= 3;
			END_IF

		3:
			SC_StoperVratDopravnika.StepName:='3 - Inicializacia - hladanie paletky';
			SC_StoperVratDopravnika.IdleTime.PT:= T#5s;
			SC_StoperVratDopravnika.AlarmTime.PT:= T#5s;
			SC_StoperVratDopravnika.IdleTime.IN:= TRUE;

			IF StoperVratDopravnika.IN.PritomnostPaletky_IS14 THEN
				StoperVratDopravnika.STAV.PoINIT:= TRUE;
				SC_StoperVratDopravnika.ResetStep:= TRUE;
				SC_StoperVratDopravnika.Step:= 101;
			ELSIF SC_StoperVratDopravnika.IdleTime.Q THEN
				StoperVratDopravnika.STAV.PoINIT:= TRUE;
				SC_StoperVratDopravnika.ResetStep:= TRUE;
				SC_StoperVratDopravnika.Step:= 100;
			END_IF

			//********************************************************Automatický režim****************************************************************************//
		100:
			SC_StoperVratDopravnika.StepName:='100 - Automaticky Rezim - cakam na príchod paletky na stoper';
			SC_StoperVratDopravnika.IdleTime.PT:= T#200ms;
			SC_StoperVratDopravnika.AlarmTime.PT:= T#5s;

			SC_StoperVratDopravnika.IdleTime.IN:= StoperVratDopravnika.IN.PritomnostPaletky_IS14;

			IF StoperVratDopravnika.KoniecCyklu AND NOT VstupVytah.Automat THEN
				SC_StoperVratDopravnika.ResetStep:= TRUE;
				SC_StoperVratDopravnika.Step:= 0;
			ELSIF SC_StoperVratDopravnika.IdleTime.Q THEN
				SC_StoperVratDopravnika.ResetStep:= TRUE;
				SC_StoperVratDopravnika.Step:= 101;
			END_IF

		101:
			SC_StoperVratDopravnika.StepName:='101 - Automaticky Rezim - cakam na vyvezenie paletky na dopravnik vstupneho vytahu';
			SC_StoperVratDopravnika.IdleTime.PT:= T#200ms;
			SC_StoperVratDopravnika.AlarmTime.PT:= T#5s;

			IF StoperVratDopravnika.KoniecCyklu AND NOT VstupVytah.Automat THEN
				SC_StoperVratDopravnika.ResetStep:= TRUE;
				SC_StoperVratDopravnika.Step:= 0;
			ELSIF SC_VstupVytah.Step = 105 AND NOT VstupVytah.IN.PritomnostPaletky_IS3 THEN
				SC_StoperVratDopravnika.ResetStep:= TRUE;
				SC_StoperVratDopravnika.Step:= 105;
			END_IF

		105:
			SC_StoperVratDopravnika.StepName:='105 - Automaticky Rezim - vyvazam paletku na dopravnik vstupneho vytahu';
			SC_StoperVratDopravnika.IdleTime.PT:= T#4s;
			SC_StoperVratDopravnika.AlarmTime.PT:= T#10s;

			IF NOT SC_StoperVratDopravnika.Switch1 THEN
				StoperVratDopravnika.OUT.StoperZASUN_YV012:= TRUE;
				SC_StoperVratDopravnika.AlarmTime.IN:= TRUE;
				SC_StoperVratDopravnika.Switch1:= TRUE;
			END_IF

			IF NOT StoperVratDopravnika.IN.PritomnostPaletky_IS14 THEN
				StoperVratDopravnika.OUT.StoperZASUN_YV012:= FALSE;
				SC_StoperVratDopravnika.AlarmTime.IN:= FALSE;
			END_IF

			IF VstupVytah.IN.PritomnostPaletky_IS3 AND NOT StoperVratDopravnika.OUT.StoperZASUN_YV012 THEN
				SC_StoperVratDopravnika.ResetStep:= TRUE;
				SC_StoperVratDopravnika.Step:= 100;
			ELSIF SC_StoperVratDopravnika.AlarmTime.Q THEN
				Alarmy[41]:= TRUE;
				PoruchaVstupnehoVytahu:= TRUE;
				SC_StoperVratDopravnika.ResetStep:= TRUE;
				SC_StoperVratDopravnika.Step:= 0;
			END_IF

			//*******************************************************Manuálny režim*******************************************************************************//
		700:
			SC_StoperVratDopravnika.StepName:='700 - Manualny Rezim';
			SC_StoperVratDopravnika.IdleTime.PT:= T#8s;
			SC_StoperVratDopravnika.AlarmTime.PT:= T#5s;

	END_CASE

END_PROGRAM

PROGRAM _EXIT
	(* Insert code here *)

END_PROGRAM
```

### Program Logical/Program/VratnyDopravnik (IEC)

#### Main.st - Init, cyclic, exit code
```iecst
PROGRAM _INIT
	(* Insert code here *)

END_PROGRAM

PROGRAM _CYCLIC

	//Volanie funkcie SequenceControl//
	SequenceControl(SC:= SC_VratnyDopravnik);

	//Reset sekcie //
	IF VratnyDopravnik.Reset THEN
		SC_VratnyDopravnik.Step:= 0;
		VratnyDopravnik.Reset:= FALSE;
	ELSIF NOT Safety.STAV.ZonaCS_AKTIVNA THEN
		SC_VratnyDopravnik.Step:= 0;
	END_IF

	CASE SC_VratnyDopravnik.Step OF

		0:
			SC_VratnyDopravnik.StepName:='0 - Nulovanie';
			VratnyDopravnik.Automat:= FALSE;
			VratnyDopravnik.KoniecCyklu:= FALSE;
			VratnyDopravnik.Manual:= FALSE;
			VratnyDopravnik.STAV.PoINIT:= FALSE;
			VratnyDopravnik.OUT.Dopravnik_ChodVPRED_ELR2:= FALSE;

			IF Safety.STAV.ZonaCS_AKTIVNA AND Linka.IN.TlakVzduchu_OK_S2 AND NOT NastalaPorucha AND Linka.STAV.Hardware_OK THEN
				SC_VratnyDopravnik.ResetStep:= TRUE;
				SC_VratnyDopravnik.Step:= 1;
			END_IF

		1:
			SC_VratnyDopravnik.StepName:='1 - Cakam na spustenie vyroby';
			VratnyDopravnik.KoniecCyklu:= FALSE;
			IF VratnyDopravnik.Automat THEN
				SC_VratnyDopravnik.Step:= 2;
			ELSIF VratnyDopravnik.Manual THEN
				SC_VratnyDopravnik.Step:= 700;
			END_IF

			//********************************************************Inicializácia****************************************************************************//

		2:
			SC_VratnyDopravnik.StepName:='2 - Inicializacia - cakam na spustenie inicializacie';
			SC_VratnyDopravnik.IdleTime.PT:= T#500ms;
			SC_VratnyDopravnik.AlarmTime.PT:= T#5s;

			SC_VratnyDopravnik.IdleTime.IN:= TRUE;

			IF SC_VratnyDopravnik.IdleTime.Q THEN
				SC_VratnyDopravnik.ResetStep:= TRUE;
				SC_VratnyDopravnik.Step:= 5;
			END_IF

		5:
			SC_VratnyDopravnik.StepName:='5 - Inicializacia - spustenie dopravnika a ukoncenie inicializacie';
			SC_VratnyDopravnik.IdleTime.PT:= T#2s;
			SC_VratnyDopravnik.AlarmTime.PT:= T#5s;

			IF NOT SC_VratnyDopravnik.Switch1 THEN
				VratnyDopravnik.OUT.Dopravnik_ChodVPRED_ELR2:= TRUE;
				SC_VratnyDopravnik.IdleTime.IN:= TRUE;
				SC_VratnyDopravnik.Switch1:= TRUE;
			END_IF

			IF SC_VratnyDopravnik.IdleTime.Q THEN
				VratnyDopravnik.STAV.PoINIT:= TRUE;
				SC_VratnyDopravnik.ResetStep:= TRUE;
				SC_VratnyDopravnik.Step:= 100;
			END_IF

			//********************************************************Automatický režim****************************************************************************//

		100:
			SC_VratnyDopravnik.StepName:='100 - Automaticky Rezim - cakam na vypnutie dopravnika';
			SC_VratnyDopravnik.IdleTime.PT:= T#200ms;
			SC_VratnyDopravnik.AlarmTime.PT:= T#5s;

			VratnyDopravnik.OUT.Dopravnik_ChodVPRED_ELR2:= NOT Linka.STAV.Dopravniky_PAUZA;

			IF VratnyDopravnik.KoniecCyklu AND NOT StoperVratDopravnika.Automat AND NOT VstupVytah.Automat AND NOT VystupVytah.Automat THEN
				SC_VratnyDopravnik.ResetStep:= TRUE;
				SC_VratnyDopravnik.Step:= 0;
			END_IF

			//*******************************************************Manuálny režim*******************************************************************************//
		700:
			SC_VratnyDopravnik.StepName:='700 - Manualny Rezim';
			SC_VratnyDopravnik.IdleTime.PT:= T#8s;
			SC_VratnyDopravnik.AlarmTime.PT:= T#5s;

	END_CASE

END_PROGRAM

PROGRAM _EXIT
	(* Insert code here *)

END_PROGRAM
```

### Program Logical/Program/Alarmy (IEC)

#### Main.st - Init, cyclic, exit code
```iecst
PROGRAM _INIT
	(* Insert code here *)

END_PROGRAM

PROGRAM _CYCLIC

    //Alarmy pracoviska (0 - 100)//
	//A0 - Porucha prepatovej ochrany !!!
	//A1 - Porucha tlaku vzduchu !!!
    //A2 - Porucha komunikacie s robotom !!!
	//A3 - Porucha komunikacie so smart kamerou !!!
	//A4 - Porucha komunikacie s modulom citaciek RFID !!!
	//A5 - Porucha komunikacie s ventilovym terminalom !!!
	//A6 - Porucha komunikacie s frekvencnymi menicmi !!!
    //A7 - Porucha PLC karty AB2 - Profinet master !!!
    //A8 - Porucha PLC karty AB3 - Safety master !!!
	//A9 - Porucha PLC karty AB4 - Safety vstupy !!!
    //A10 - Porucha PLC karty AB5 - Digitalne vstupy !!!
    //A11 - Porucha PLC karty AB6 - Digitalne vstupy !!!
    //A12 - Porucha PLC karty AB7 - Digitalne vstupy !!!
	//A13 - Porucha PLC karty AB8 - Digitalne vystupy !!!
	//A14 - Porucha PLC karty AB9 - Digitalne vystupy !!!
	//A15 - Porucha PLC karty AB10 - X2X master !!!
	//A16 - Porucha modulu DI1 - Digitalne vstupy !!!
	//A17 - Porucha modulu DI2 - Digitalne vstupy !!!
	//A18 - Porucha modulu DI3 - Digitalne vstupy !!!
	//A19 - Porucha modulu SI1 - Safety vstupy !!!
	//A20 - Porucha modulu SI2 - Safety vstupy !!!
	//A21 -
	//A22 -
	//A23 -
	//A24 -
	//A25 -
	//A26 -
	//A27 -
	//A28 -
	//A29 -
	//A30 -
    //A31 - Bolo stlacene tlacitko CS robota !!!
    //A32 - Bolo stlacene tlacitko CS ovladacieho panela !!!
	//A33 - Bolo stlacene tlacitko CS vstupneho vytahu !!!
	//A34 - Bolo stlacene tlacitko CS vystupneho vytahu !!!
	//A35 - Porucha vyvezenia paletky zo stopra pred cistenim !!!
	//A36 - Porucha spustenia cistenia !!!
	//A37 - Porucha otacania hornej trisky cistenia !!!
	//A38 - Porucha otacania spodnej trisky cistenia !!!
	//A39 - Porucha vyvezenia paletky zo stopra po cisteni !!!
    //A40 - Porucha vyvezenia paletky zo stopra vystupneho dopravnika !!!
	//A41 - Porucha vyvezenia paletky zo stopra vratneho dopravnika !!!
	//A42 - Porucha otvorenia dveri vstupneho vytahu !!!
	//A43 - Porucha zatvorenia dveri vstupneho vytahu !!!
	//A44 - Pritomnost paletky na prechode medzi vstupnym vytahom a dopravnikom !!!
	//A45 - Porucha navazania paletky na dopravnik vstupneho vytahu !!!
	//A46 - Narusenie optickej bariery vstupneho vytahu !!!
	//A47 - Paletka v koliznej pozicii vstupneho vytahu !!!
	//A48 - Porucha vyvezenia paletky z dopravnika vstupneho vytahu !!!
	//A49 - Pritomnost paletky na prechode medzi vystupnym vytahom a dopravnikom !!!
	//A50 - Narusenie optickej bariery vystupneho vytahu !!!
	//A51 - Paletka v koliznej pozicii vystupneho vytahu !!!
	//A52 - Porucha navazania paletky na dopravnik vystupneho vytahu !!!
	//A53 - Porucha zdvihu centrovania paletky na pozicii etiketovania !!!
	//A54 - Porucha zasunutia centrovania paletky na pozicii etiketovania !!!
	//A55 - Porucha vytlacenia etikety !!!
	//A56 - Porucha vyvezenia paletky zo stopra etiketovania !!!
	//A57 - Porucha zdvihu centrovania paletky na pozicii stopra dopravnika NG !!!
	//A58 - Porucha zasunutia centrovania paletky na pozicii stopra dopravnika NG !!!
	//A59 - Porucha presunu centrovania paletky do strednej polohy na pozicii stopra dopravnika NG !!!
	//A60 - Porucha precitania cisla paletky na pozicii vstupneho vytahu !!!
	//A61 - Porucha precitania cisla paletky na pozicii stopra etiketovania !!!
	//A62 - Porucha precitania cisla paletky na pozicii vystupneho vytahu !!!
	//A63 - Porucha vyvezenia paletky na dopravnik NG !!!
	//A64 - Porucha navezenia paletky z dopravnika NG !!!
	//A65 - Porucha vyvezenia paletky zo stopra dopravnika NG !!!
	//A66 - Porucha precitania QR kodu interneho stitku na pozicii stopra etiketovania !!!
	//A67 - Porucha menica zdvihu vstupneho vytahu !!!
	//A68 - Porucha menica pohonu dopravnika cistenia !!!
	//A69 - Porucha menica zdvihu vystupneho vytahu !!!
	//A70 - Porucha precitania cisla paletky na pozicii dopravnika cistenia !!!
	//A71 - Porucha, nepovolene otvorenie servisnych dveri tlaciarne !!!
	//A72 - Narusenie optickej bariery dopravnika NG !!!
	//A73 - Bol zastaveny program robota !!!
	//A74 - Porucha komunikácie so serverom Panasonic !!!
	//A75 - Kamera robota nieje READY !!!
	//A76 - Porucha odobratia etikety z tlačiarne !!!

     //***********************************Hladanie poruchy*****************************************//

	FOR a:=0 TO 100 BY 1 DO
		Alarmy[a];
		IF Alarmy[a] = TRUE THEN
			NastalaPorucha:= TRUE;
		END_IF
	END_FOR

	//********************************Zobrazenie symbolu alarmu*****************************************************//

	IF NastalaPorucha THEN
		Vizu.ZobrazSymbolAlarmu:= Blikac500ms;
	ELSE
		Vizu.ZobrazSymbolAlarmu:= FALSE;
	END_IF

	//*************************************Potvrdenie alarmov*********************************************************//
	IF PotvrdenieAlarmov THEN
		brsmemset(ADR(Alarmy),0,SIZEOF(Alarmy));
		NastalaPorucha:= FALSE;
		PoruchaBunky:= FALSE;
		PoruchaCistenia:= FALSE;
		PoruchaLinky:= FALSE;
		PoruchaVstupnehoVytahu:= FALSE;
		PoruchaVystupnehoVytahu:= FALSE;
		Linka.STAV.PoruchaOtacaniaTrysiek:= FALSE;
		Linka.Majak_HukackaON:= FALSE;
		IF VstupVytah.MenicZdvihu_FM2.STAV.PORUCHA THEN
			VstupVytah.MenicZdvihu_FM2.CMD.Potvrd_PORUCHU:= TRUE;
		END_IF
		IF VystupVytah.MenicZdvihu_FM3.STAV.PORUCHA THEN
			VystupVytah.MenicZdvihu_FM3.CMD.Potvrd_PORUCHU:= TRUE;
		END_IF
		IF DopravCistenia.MenicDopravnika_FM1.STAV.PORUCHA THEN
			DopravCistenia.MenicDopravnika_FM1.CMD.Potvrd_PORUCHU:= TRUE;
		END_IF
		PotvrdenieAlarmov:= FALSE;
	END_IF

	//*******************************Porucha prepatovej ochrany*********************************************************//
	IF Safety.STAV.ZonaCS_AKTIVNA AND NOT Linka.IN.PrepatovaOchrana_OK THEN
		Alarmy[0]:= TRUE;
	END_IF

	//*******************************Porucha tlaku vzduchu**************************************************************//
	CasKontrolyTlakuVzduchu.IN:= Safety.STAV.ZonaCS_AKTIVNA AND NOT Linka.IN.TlakVzduchu_OK_S2;

	IF CasKontrolyTlakuVzduchu.Q THEN
		Alarmy[1]:= TRUE;
		PoruchaLinky:= TRUE;
	END_IF

	CasKontrolyTlakuVzduchu.PT:= T#2s;
	CasKontrolyTlakuVzduchu();

	//********************************Porucha komunikácie s robotom******************************************************//
	CasKontroly_KOM_Robota.IN:= Safety.STAV.ZonaCS_AKTIVNA AND NOT StavHardware.Komunikacia_Robot_OK;
	IF CasKontroly_KOM_Robota.Q THEN
		Alarmy[2]:= TRUE;
		PoruchaBunky:= TRUE;
	END_IF

	CasKontroly_KOM_Robota.PT:= T#2s;
	CasKontroly_KOM_Robota();

	//********************************Porucha komunikácie s kamerou******************************************************//
	CasKontroly_KOM_Kamery.IN:= Robot.Automat AND NOT StavHardware.Komunikacia_Kamera_OK;
	IF CasKontroly_KOM_Kamery.Q THEN
		Alarmy[3]:= TRUE;
		PoruchaBunky:= TRUE;
	END_IF

	CasKontroly_KOM_Kamery.PT:= T#1s;
	CasKontroly_KOM_Kamery();

	//********************************Porucha komunikácie s modulom RFID čitačiek******************************************************//
	CasKontroly_KOM_IOlinkModulu.IN:= Safety.STAV.ZonaCS_AKTIVNA AND NOT StavHardware.Komunikacia_RFIDModul_OK;
	IF CasKontroly_KOM_RFIDModulu.Q THEN
		Alarmy[4]:= TRUE;
		PoruchaLinky:= TRUE;
	END_IF

	CasKontroly_KOM_RFIDModulu.PT:= T#2s;
	CasKontroly_KOM_IOlinkModulu();

	//********************************Porucha komunikácie s ventilovým terminálom******************************************************//
	CasKontroly_KOM_VentTerminalu.IN:= Safety.STAV.ZonaCS_AKTIVNA AND NOT StavHardware.Komunikacia_VentTerminal_OK;
	//	IF CasKontroly_KOM_VentTerminalu.Q THEN
	//		Alarmy[5]:= TRUE;
	//		PoruchaLinky:= TRUE;
	//	END_IF

	CasKontroly_KOM_VentTerminalu.PT:= T#2s;
	CasKontroly_KOM_VentTerminalu();

	//********************************Porucha komunikácie s frekvenčnými meničmy******************************************************//
	CasKontroly_KOM_MenicovFM.IN:= Safety.STAV.ZonaCS_AKTIVNA AND NOT StavHardware.Komunikacia_MeniceFM_OK;
	IF CasKontroly_KOM_MenicovFM.Q THEN
		Alarmy[6]:= TRUE;
		PoruchaLinky:= TRUE;
	END_IF

	CasKontroly_KOM_MenicovFM.PT:= T#2s;
	CasKontroly_KOM_MenicovFM();

	//**********************************Porucha - karty PLC niesu online**************************************************//
	IF CasKontroly_KarietPLC.Q THEN
		IF NOT StavHardware.KartaAB2_ProfinetMaster_OK THEN
			Alarmy[7]:= TRUE;
			PoruchaLinky:= TRUE;
		END_IF
		IF NOT StavHardware.KartaAB3_SafetyMaster_OK THEN
			Alarmy[8]:= TRUE;
			PoruchaLinky:= TRUE;
		END_IF
		IF NOT StavHardware.KartaAB4_SafetyDI_OK THEN
			Alarmy[9]:= TRUE;
			PoruchaLinky:= TRUE;
		END_IF
		IF NOT StavHardware.KartaAB5_16DI_OK THEN
			Alarmy[10]:= TRUE;
			PoruchaLinky:= TRUE;
		END_IF
		IF NOT StavHardware.KartaAB6_16DI_OK THEN
			Alarmy[11]:= TRUE;
			PoruchaLinky:= TRUE;
		END_IF
		IF NOT StavHardware.KartaAB7_16DI_OK THEN
			Alarmy[12]:= TRUE;
			PoruchaLinky:= TRUE;
		END_IF
		IF NOT StavHardware.KartaAB8_16DO_OK THEN
			Alarmy[13]:= TRUE;
			PoruchaLinky:= TRUE;
		END_IF
		IF NOT StavHardware.KartaAB9_16DO_OK THEN
			Alarmy[14]:= TRUE;
			PoruchaLinky:= TRUE;
		END_IF
		IF NOT StavHardware.KartaAB10_X2X_OK THEN
			Alarmy[15]:= TRUE;
			PoruchaLinky:= TRUE;
		END_IF
		IF NOT StavHardware.ModulDI1_16DI_OK THEN
			Alarmy[16]:= TRUE;
			PoruchaLinky:= TRUE;
		END_IF
		IF NOT StavHardware.ModulDI2_16DI_OK THEN
			Alarmy[17]:= TRUE;
			PoruchaLinky:= TRUE;
		END_IF
		IF NOT StavHardware.ModulDI3_8DI_OK THEN
			Alarmy[18]:= TRUE;
			PoruchaLinky:= TRUE;
		END_IF
		IF NOT StavHardware.ModulSI1_4SI_OK THEN
			Alarmy[19]:= TRUE;
			PoruchaLinky:= TRUE;
		END_IF
		IF NOT StavHardware.ModulSI2_4SI_OK THEN
			Alarmy[20]:= TRUE;
			PoruchaLinky:= TRUE;
		END_IF
		IF NOT StavHardware.Komunikacia_Panasonic_OK THEN
			Alarmy[74]:= TRUE;
			PoruchaLinky:= TRUE;
		END_IF
	END_IF

	IF Safety.STAV.ZonaCS_AKTIVNA AND NOT Linka.STAV.Hardware_OK THEN
		CasKontroly_KarietPLC.IN:= TRUE;
	ELSE
		CasKontroly_KarietPLC.IN:= FALSE;
	END_IF

	CasKontroly_KarietPLC.PT:= T#2s;
	CasKontroly_KarietPLC();

	//**********************************Porucha bolo stlacene tlačítko CS robota***************************************//
	IF EDGENEG(Safety.STAV.CS_Robot_Odblokovany) THEN
		Alarmy[31]:= TRUE;
		PoruchaLinky;
	END_IF

	//**********************************Porucha bolo stlacene tlačítko CS ovládacieho panela***************************************//
	IF EDGENEG(Safety.STAV.CS_OvlPanel_Odblokovany) THEN
		Alarmy[32]:= TRUE;
		PoruchaLinky;
	END_IF

	//**********************************Porucha bolo stlacene tlačítko CS vstupného výťahu***************************************//
	IF EDGENEG(Safety.STAV.CS_VstupnyVytah_Odblokovany) THEN
		Alarmy[33]:= TRUE;
		PoruchaLinky;
	END_IF

	//**********************************Porucha bolo stlacene tlačítko CS výstupného výťahu***************************************//
	IF EDGENEG(Safety.STAV.CS_VystupnyVytah_Odblokovany) THEN
		Alarmy[34]:= TRUE;
		PoruchaLinky;
	END_IF

	//************************************Porucha meniča zdvihu vstupného výťahu***************************************************//
	IF VstupVytah.Automat AND VstupVytah.MenicZdvihu_FM2.STAV.PORUCHA THEN
		Alarmy[67]:= TRUE;
		PoruchaVstupnehoVytahu:= TRUE;
	END_IF

	//************************************Porucha meniča pohonu dopravníka čistenia***************************************************//
	IF DopravCistenia.Automat AND DopravCistenia.MenicDopravnika_FM1.STAV.PORUCHA THEN
		Alarmy[68]:= TRUE;
		PoruchaCistenia:= TRUE;
	END_IF

	//************************************Porucha meniča zdvihu výstupného výťahu***************************************************//
	IF VystupVytah.Automat AND VystupVytah.MenicZdvihu_FM3.STAV.PORUCHA THEN
		Alarmy[69]:= TRUE;
		PoruchaVystupnehoVytahu:= TRUE;
	END_IF

END_PROGRAM

PROGRAM _EXIT
	(* Insert code here *)

END_PROGRAM
```

#### Variables.var - Local variables
```iecst
VAR
	a : USINT := 0;
	CasKontroly_KarietPLC : TON;
	CasKontroly_KOM_Robota : TON;
	CasKontroly_TlakuVzduchu : TON := (0);
	CasKontroly_KOM_VentTerminalu : TON := (0);
	CasKontroly_KOM_IOlinkModulu : TON := (0);
	CasKontroly_KOM_Kamery : TON := (0);
	CasKontroly_KOM_MenicovFM : TON := (0);
	CasKontrolyTlakuVzduchu : TON;
	CasKontroly_KOM_RFIDModulu : TON;
END_VAR
```

### Program Logical/Program/StatistikaLinky (IEC)

#### Main.st - Init, cyclic, exit code
```iecst
PROGRAM _INIT
	VstupnyVytah_Statistika.IN.TaskovaTrieda_ms:= 2;
	StoperPredCistenim_Statistika.IN.TaskovaTrieda_ms:= 2;
	StoperPoCisteni_Statistika.IN.TaskovaTrieda_ms:= 2;
	StoperEtiketovania_Statistika.IN.TaskovaTrieda_ms:= 2;
	StoperDopravNG_Statistika.IN.TaskovaTrieda_ms:= 2;
	VystupnyVytah_Statistika.IN.TaskovaTrieda_ms:= 2;
	Linka_Statistika.IN.TaskovaTrieda_ms:= 2;
END_PROGRAM

PROGRAM _CYCLIC

	VstupnyVytah_Statistika();
	StoperPredCistenim_Statistika();
	StoperPoCisteni_Statistika();
	StoperEtiketovania_Statistika();
	StoperDopravNG_Statistika();
	VystupnyVytah_Statistika();
	Linka_Statistika();

	//********************************************Meranie taktime vstupného výťahu*****************************************************//
	IF VstupnyVytah_Statistika.IN.ZAPIS_MeraniaCasu AND VstupnyVytah_Statistika.OUT.Stav_ZapisCasu_DONE THEN
		VstupnyVytah_Statistika.IN.ZAPIS_MeraniaCasu:= FALSE;
	END_IF

	//Zobrazenie štatistik//
	VstupnyVytah_Statistika.OUT.NameranyCas_v_Sekundach;

	//Reset priemerného času//
	IF VstupnyVytah_Statistika.IN.RESET_HistorieMeraniCasu AND VstupnyVytah_Statistika.OUT.Stav_RESET_HistorieMerani_DONE THEN
		VstupnyVytah_Statistika.IN.RESET_HistorieMeraniCasu:= FALSE;
	END_IF

	//***********************************************Meranie taktime stopra pred čistením******************************************************//
	IF StoperPredCistenim_Statistika.IN.ZAPIS_MeraniaCasu AND StoperPredCistenim_Statistika.OUT.Stav_ZapisCasu_DONE THEN
		StoperPredCistenim_Statistika.IN.ZAPIS_MeraniaCasu:= FALSE;
	END_IF

	//Zobrazenie štatistik//
	StoperPredCistenim_Statistika.OUT.NameranyCas_v_Sekundach;

	//Reset priemerného času//
	IF StoperPredCistenim_Statistika.IN.RESET_HistorieMeraniCasu AND StoperPredCistenim_Statistika.OUT.Stav_RESET_HistorieMerani_DONE THEN
		StoperPredCistenim_Statistika.IN.RESET_HistorieMeraniCasu:= FALSE;
	END_IF

	//********************************************Meranie taktime stopra po čistení***********************************************************//
	IF StoperPoCisteni_Statistika.IN.ZAPIS_MeraniaCasu AND StoperPoCisteni_Statistika.OUT.Stav_ZapisCasu_DONE THEN
		StoperPoCisteni_Statistika.IN.ZAPIS_MeraniaCasu:= FALSE;
	END_IF

	//Zobrazenie štatistik//
	StoperPoCisteni_Statistika.OUT.NameranyCas_v_Sekundach;

	//Reset priemerného času//
	IF StoperPoCisteni_Statistika.IN.RESET_HistorieMeraniCasu AND StoperPoCisteni_Statistika.OUT.Stav_RESET_HistorieMerani_DONE THEN
		StoperPoCisteni_Statistika.IN.RESET_HistorieMeraniCasu:= FALSE;
	END_IF

	//********************************************Meranie taktime stopra etiketovania***************************************************************//
	IF StoperEtiketovania_Statistika.IN.ZAPIS_MeraniaCasu AND StoperEtiketovania_Statistika.OUT.Stav_ZapisCasu_DONE THEN
		StoperEtiketovania_Statistika.IN.ZAPIS_MeraniaCasu:= FALSE;
	END_IF

	//Zobrazenie štatistik//
	StoperEtiketovania_Statistika.OUT.NameranyCas_v_Sekundach;

	//Reset priemerného času//
	IF StoperEtiketovania_Statistika.IN.RESET_HistorieMeraniCasu AND StoperEtiketovania_Statistika.OUT.Stav_RESET_HistorieMerani_DONE THEN
		StoperEtiketovania_Statistika.IN.RESET_HistorieMeraniCasu:= FALSE;
	END_IF

	//*********************************Meranie taktime stopra dopravníka NG*******************************************************************//
	IF StoperDopravNG_Statistika.IN.ZAPIS_MeraniaCasu AND StoperDopravNG_Statistika.OUT.Stav_ZapisCasu_DONE THEN
		StoperDopravNG_Statistika.IN.ZAPIS_MeraniaCasu:= FALSE;
	END_IF

	//Zobrazenie štatistik//
	StoperDopravNG_Statistika.OUT.NameranyCas_v_Sekundach;

	//Reset priemerného času//
	IF StoperDopravNG_Statistika.IN.RESET_HistorieMeraniCasu AND StoperDopravNG_Statistika.OUT.Stav_RESET_HistorieMerani_DONE THEN
		StoperDopravNG_Statistika.IN.RESET_HistorieMeraniCasu:= FALSE;
	END_IF

	//*********************************************Meranie taktime výstupného výťahu****************************************************************//
	IF VystupnyVytah_Statistika.IN.ZAPIS_MeraniaCasu AND VystupnyVytah_Statistika.OUT.Stav_ZapisCasu_DONE THEN
		VystupnyVytah_Statistika.IN.ZAPIS_MeraniaCasu:= FALSE;
	END_IF

	//Zobrazenie štatistik//
	VystupnyVytah_Statistika.OUT.NameranyCas_v_Sekundach;

	//Reset priemerného času//
	IF VystupnyVytah_Statistika.IN.RESET_HistorieMeraniCasu AND VystupnyVytah_Statistika.OUT.Stav_RESET_HistorieMerani_DONE THEN
		VystupnyVytah_Statistika.IN.RESET_HistorieMeraniCasu:= FALSE;
	END_IF

	//Reset počtu kusov OK a NG//
	IF RESET_PoctuVyrobenychKusov THEN
		PocetVyrobenychKusov_OK:= 0;
		PocetVyrobenychKusov_NG:= 0;
		Pomer_OK_kusov_IDR:= 0;
		RESET_PoctuVyrobenychKusov:= FALSE;
	END_IF

	//Vyrátanie IDR percentuálny pomer kusov OK k celkovému počtu vyrobených kusov//
	IF PocetVyrobenychKusov_OK <> 0 THEN
		Pomer_OK_kusov_IDR:= 100 * (PocetVyrobenychKusov_OK/(PocetVyrobenychKusov_OK + PocetVyrobenychKusov_NG));
	END_IF

	//Reset celkového počtu kusov//
	IF RESET_CelkovehoPoctuKusov THEN
		CelkovyPocetVyrobenychKusov:= 0;
		RESET_CelkovehoPoctuKusov:= FALSE;
	END_IF

END_PROGRAM

PROGRAM _EXIT
	(* Insert code here *)

END_PROGRAM
```

### Program Logical/Program/IonizacnaJednotka (IEC)
